(* CODESYS project TC_lib_v0-0-0-1.library
   Company: RWTH
   Title: Tc_Wilo_LIB
   Placeholder: Tc_Wilo_LIB
   Author: Vonnahme
   Version: 0.0.0.1

Project tree, tasks and I/O mapping:
  libraries: Tc2_Standard, * (Beckhoff Automation GmbH); Tc2_System, * (Beckhoff Automation GmbH); Tc2_TcpIp, * (Beckhoff Automation GmbH); Tc2_Utilities, * (Beckhoff Automation GmbH); Tc3_Interfaces, * (Beckhoff Automation GmbH); Tc3_Module, * (Beckhoff Automation GmbH)
  ADS/
    function block FB_ADS_READ [ST]
    function block FB_ADS_WRITE [ST]
  CAN/
    Definitions/
      data type eBusCommand
      data type eBusControlMode
      data type eEffCommand
      data type SDO_Datapoint
      data type StratosControl
      data type WILO_Stratos
      data type WILO_StratosGiga_IPE
    Stratos/
      function block FB_Stratos_CAN [ST]
    StratosGiga_IPE/
      function block FB_StratosGIGA_IPE [ST]
    function block FB_SDO_READ [ST]
    function block FB_SDO_READ_v0 [ST]
    function block FB_SDO_WRITE [ST]
  Datenlogger/
    Definitions/
      data type Log_Datapoint
      data type Log_Struct_HMI
    FB/
      function block FB_FILE [ST]
      function block FB_FOLDER [ST]
      function block FB_LOGGING [ST]
      function block FB_TIME [ST]
    function block FB_Datenlogger [ST]
  Functions/
    function FUN_ByteArrToString [ST]
    function FUN_DatatypSize [ST]
    function FUN_StringToByteArr [ST]
    function SCALE [ST]
  Timetable/
    DUT/
      data type Struct_TimeTable
    function block FB_TimeTable [ST]
  TypeDef/
    data type Datatyp
  Version/
    global variables Global_Version
*)

// CAN/Definitions/eBusCommand
{attribute 'qualified_only'}
{attribute 'strict'}
TYPE eBusCommand : 
(
	RemoteOn:=97,
	RemoteOff:=96
);
END_TYPE

// CAN/Definitions/eBusControlMode
{attribute 'qualified_only'}
//{attribute 'strict'}
TYPE eBusControlMode : 
(
	nc:=0,
	dpc:=5,
	dpv:=6
);
END_TYPE

// CAN/Definitions/eEffCommand
{attribute 'qualified_only'}
//{attribute 'strict'}
TYPE eEffCommand : 
(
	PumpOn:=1,
	PumpOff:=0,
	RemoteOn:=97,
	RemoteOff:=96
);
END_TYPE

// CAN/Definitions/SDO_Datapoint
TYPE SDO_Datapoint :
STRUCT
	sDatapointNo		:STRING;
	sDescription 		:STRING;
	sValue				:STRING;
	eDatatyp			:Datatyp;
	sUnit				:STRING;
	bReadSuccesfull		:BOOL;
END_STRUCT
END_TYPE

// CAN/Definitions/StratosControl
TYPE StratosControl :
STRUCT
		eBusCommand								:eBusCommand;		// PumpOn, PumpOff
		eBusControlMode							:eBusControlMode;	// nc,dpc, dpv
		nBusSetpoint							:LREAL;			//[%,rpm,mWs]
END_STRUCT
END_TYPE

// CAN/Definitions/WILO_Stratos
TYPE WILO_Stratos :
STRUCT
	arrPumpInformation						:ARRAY [1..100] OF SDO_Datapoint;
	iSpeed									:UINT;				//[rpm]	
	nPressure								:LREAL;				//[mWs]
	nFlow									:LREAL;				//[m³/h]		
	nInputPower								:LREAL;				//[W]
	nConsumption							:LREAL;				//[kWh]	
	nMediumTemp								:LREAL;				//[°C]
	nOperatingHours							:LREAL;				//[h]		
	eEff_Command							:eEffCommand;	
	eEff_ControlMode						:eBusControlMode;	
	nEff_Setpoint							:LREAL;				//[%]
	nEff_Setpoint_abs						:LREAL;				//[rpm, mWs]
	eSel_Command							:eEffCommand;
	eSel_ControlMode						:eBusControlMode;	
	nSel_Setpoint							:LREAL;				//[%]
	nSel_Setpoint_abs						:LREAL;				//[rpm, mWs]
	iPumpType								:UINT;				//[PumpType]	
	nMaxValue								:LREAL;				//[mWs], [rpm]
	nMinValue								:LREAL;				//[mWs], [rpm]
	iCurrentWarning							:USINT;				//[Error Code]	
	eBusCommand								:eBusCommand;
	eBusControlMode							:eBusControlMode;
	nBusSetpoint							:LREAL;		
END_STRUCT
END_TYPE

// CAN/Definitions/WILO_StratosGiga_IPE
TYPE WILO_StratosGiga_IPE :
STRUCT
	arrPumpInformation						:ARRAY [1..100] OF SDO_Datapoint;
	iSpeed									:UINT;				//[rpm]	
	nPressure								:LREAL;				//[mWs]
	nFlow									:LREAL;				//[m³/h]		
	nInputPower								:LREAL;				//[W]
	nConsumption							:LREAL;				//[kWh]	
	iPressureSensorSource					:USINT;				// 2 Pump Housing, 3 External, 5 LON
	nOperatingHours							:LREAL;				//[h]		
	eEff_Command							:eEffCommand;	
	eEff_ControlMode						:eBusControlMode;	
	nEff_Setpoint							:LREAL;				//[%]
	nEff_Setpoint_abs						:LREAL;				//[rpm, mWs]
	eSel_Command							:eEffCommand;
	eSel_ControlMode						:eBusControlMode;	
	nSel_Setpoint							:LREAL;				//[%]
	nSel_Setpoint_abs						:LREAL;				//[rpm, mWs]
	iPumpType								:UINT;				//[PumpType]	
	nMaxValue								:LREAL;				//[mWs], [rpm]
	iCurrentWarning							:USINT;				//[Error Code]	
	eBusCommand								:eBusCommand;
	eBusControlMode							:eBusControlMode;
	nBusSetpoint							:LREAL;	
	iBusStatus								:USINT;
	iControlStatus 							:USINT;
	iReadyForOperation 						:USINT;
	iPumpIsOperating 						:USINT;
	iServiceRequired 						:USINT;
	nElectricalCurrent 						:LREAL;				// [A]
	nVoltageLevel 							:LREAL;				// [V]
END_STRUCT
END_TYPE

// Datenlogger/Definitions/Log_Datapoint
TYPE Log_Datapoint :
STRUCT
	sID				:T_MaxString;
	sDescription 	:T_MaxString;
	sUnit			:T_MaxString;
	sValue 			:T_MaxString;
END_STRUCT
END_TYPE

// Datenlogger/Definitions/Log_Struct_HMI
TYPE Log_Struct_HMI :
STRUCT
	bLogging :BOOL;
	sCycleTime :STRING:='T#10s';
	sFolderPath :STRING;
	iErrors	:UINT;
	iNumberOfLoggedDatapoints :INT;
	arrLogDatapoints :ARRAY [0..499] OF Log_Datapoint;
END_STRUCT
END_TYPE

// Timetable/DUT/Struct_TimeTable
TYPE Struct_TimeTable :
STRUCT
	wDayOfWeek	:WORD:=99;		// 0= inactiv, 1=Sunday, 2=Monday, ... 7=Saturday, 8=daily, 9=Weekend, 10=Mo-Fr, 99=last row
	wHour		:WORD;
	wMinute		:WORD;
	nValue		:LREAL;
END_STRUCT
END_TYPE

// TypeDef/Datatyp
{attribute 'qualified_only'}
{attribute 'strict'}
TYPE Datatyp :
(
	_NotDefined:=0,
	_BYTE:=1,
	_WORD:=2,
	_DWORD:=3,
	_SINT:=4,
	_INT:=5,
	_DINT:=6,
	_LINT:=7,
	_USINT:=8,
	_UINT:=9,
	_UDINT:=10,
	_ULINT:=11,
	_REAL:=12,
	_LREAL:=13,
	_BOOL:=14,
	_ENUM:=15
);
END_TYPE

// Version/Global_Version
{attribute 'TcGenerated'}
// This function has been automatically generated from the project information.
VAR_GLOBAL CONSTANT
	{attribute 'const_non_replaced'}
	{attribute 'linkalways'}
	stLibVersion_Tc_Wilo_LIB : ST_LibVersion := (iMajor := 0, iMinor := 0, iBuild := 0, iRevision := 1, sVersion := '0.0.0.1');
END_VAR

// ADS/FB_ADS_READ
FUNCTION_BLOCK FB_ADS_READ
VAR_INPUT
	/// The AMSNetID addresses the FC5101 card. Can be empty if only one local single channel card is present
	ADSNetID: STRING(23);
	/// This Port No. of the Reading DataPoint 
	PortNr: WORD;
	/// hexadecimal '16x000'
	IndexGroup: DWORD;
	/// hexadecimal '16x000'
	IndexOffset: DWORD;
	/// hexadecimal '16x000'
	DataLength: DWORD;
	/// only reset to FALSE after ReadDataAvailable=TRUE
	StartReading: BOOL;
END_VAR
VAR_OUTPUT
	ReadData: ARRAY[0..255] OF BYTE;
	ReadDataAvailable: BOOL;
	Error: DWORD;
END_VAR
VAR
	state: BYTE := 0;
	ADSREAD: ADSREAD;
END_VAR

CASE state OF
0:
	IF StartReading THEN
		ReadDataAvailable := FALSE;
		Error := 0;
		ADSRead(
			NETID:= ADSNetID,
			PORT:= PortNr,
			IDXGRP:= IndexGroup,
			IDXOFFS:= IndexOffset,
			LEN:= DataLength,
			DESTADDR:= ADR(ReadData),
			READ:= TRUE,
			TMOUT := T#1s
		);
		IF ADSRead.err THEN
			state := 2;
			(*ReadDataAvailable := TRUE;*)
			Error := ADSRead.ErrId;
		ELSE
			state := 1;
		END_IF
	ELSE
		ADSRead(
			NETID:= ADSNetID,
			PORT:= PortNr,
			IDXGRP:= IndexGroup,
			IDXOFFS:= IndexOffset,
			LEN:= DataLength,
			DESTADDR:= ADR(ReadData),
			READ:= FALSE,
			TMOUT := T#1s
		);
	END_IF

1:
	ADSRead(READ:= FALSE);
	IF ADSRead.err THEN
		state := 2;
		(*ReadDataAvailable := TRUE;*)
		Error := ADSRead.ErrId;
	ELSE
		IF NOT ADSRead.busy THEN
			state := 2;
			(*ReadDataAvailable := TRUE;*)
		END_IF
	END_IF

2: 
	ADSRead(READ:= FALSE);
	ReadDataAvailable := TRUE;
	state := 0;
END_CASE

END_FUNCTION_BLOCK

// ADS/FB_ADS_WRITE
FUNCTION_BLOCK FB_ADS_WRITE
VAR_INPUT
	/// The AMSNetID addresses the FC5101 card. Can be empty if only one local single channel card is present
	ADSNetID: STRING(23);
	/// This Port No. of the Reading DataPoint 
	PortNr: WORD;
	/// hexadecimal '16x000'
	IndexGroup: DWORD;
	/// hexadecimal '16x000'
	IndexOffset: DWORD;
	/// hexadecimal '16x000'
	DataLength: DWORD;
	/// only reset to FALSE after WriteDataFinished=TRUE
	StartWriting: BOOL;
	///This array contains the data to be written to the CANopen Object Dictionary
	WriteData: ARRAY[0..255] OF BYTE;
END_VAR
VAR_OUTPUT
	WriteDataFinished: BOOL;
	Error: DWORD;
END_VAR
VAR
	state: BYTE := 0;
	ADSWRITE: ADSWRITE;
END_VAR

CASE state OF
0:
	IF StartWriting THEN
		WriteDataFinished := FALSE;
		Error := 0;
		ADSWrite(
			NETID:= ADSNetID,
			PORT:= PortNr,
			IDXGRP:= IndexGroup,
			IDXOFFS:= IndexOffset,
			LEN:= DataLength,
			SRCADDR:= ADR(WriteData),
			WRITE:= TRUE,
			TMOUT := T#1s
		);
		IF ADSWrite.err THEN
			state := 2;
			(*WriteDataFinished := TRUE;*)
			Error := ADSWrite.ErrId;
		ELSE
			state := 1;
		END_IF
	ELSE
		ADSWrite(
			NETID:= '',
			PORT:= PortNr,
			IDXGRP:= IndexGroup,
			IDXOFFS:= IndexOffset,
			LEN:= DataLength,
			SRCADDR:= ADR(WriteData),
			WRITE:= FALSE,
			TMOUT := T#1s
		);
	END_IF

1:
	ADSWrite(WRITE:= FALSE);
	IF ADSWrite.err THEN
		state := 2;
		(*WriteDataFinished := TRUE;*)
		Error := ADSWrite.ErrId;
	ELSE
		IF NOT ADSWrite.busy THEN
			state := 2;
			(*WriteDataFinished := TRUE;*)
		END_IF
	END_IF

2:
	ADSWrite(WRITE:= FALSE);
	state := 0;
	WriteDataFinished := TRUE;
END_CASE

END_FUNCTION_BLOCK

// CAN/Stratos/FB_Stratos_CAN
FUNCTION_BLOCK FB_Stratos_CAN
VAR_INPUT
	// CAN configuration
		sCAN_NetID								:STRING (23);	// NetID of CAN Master
		iCAN_NodeID								:UINT;		// NodeId (automatic calculation of Port No.
	// control configuration
		bReadOnly								:BOOL;		// deactivate pump control
		bUseAbsoluteSetpoint					:BOOL;		// use rpm or mWs instead of %
		bExternalCommandOverride				:BOOL:=TRUE;	// Use  for pump control Struct instead of PumpInformationStruct to control the pump
		stPumpControl							:StratosControl; // Struct for control pump by external PLC Code
END_VAR
VAR_OUTPUT
	// Error
		iReadError								:UINT;	// number of Errors (read)
		iWriteError								:UINT;	// number of Errors (write)
	
	// Structure	
		stPumpInformation						:WILO_Stratos; // Information (Control) of pump
			
	// Logging
		arrDatenpunkt_IDs_Pump					:ARRAY [0..99] OF T_MaxString;			(*Beschreibung der Datenpunkte*)
		arrDatenpunkt_Values_Pump				:ARRAY [0..99] OF T_MaxString;			(*Messwerte der Datenpunkte*)
		iDatapoints_Pump						:INT			:=0;
END_VAR
VAR	
	// Datapoints
(*		iSpeed									:UINT;			//[rpm]	
		nPressure								:LREAL;			//[mWs]
		nFlow									:LREAL;			//[m³/h]		
		nInputPower								:LREAL;			//[W]
		nConsumption							:LREAL;			//[kWh]	
		nMediumTemp								:LREAL;			//[°C]
		nOperatingHours							:LREAL;			//[h]		
		eEff_Command							:eEffCommand;	
		eEff_ControlMode						:eBusControlMode;	
		nEff_Setpoint							:LREAL;			//[%]
		nEff_Setpoint_abs						:LREAL;			//[rpm, mWs]
		eSel_Command							:eEffCommand;
		eSel_ControlMode						:eBusControlMode;
		nSel_Setpoint							:LREAL;			//[%]
		nSel_Setpoint_abs						:LREAL;			//[rpm, mWs]
		iPumpType								:UINT;			//[PumpType]	
		nMaxValue								:LREAL;			//[mWs], [rpm]
		iCurrentWarning							:USINT;			//[Error Code]		
*)
	// Read
		imaxValue								:UINT;	
		iminValue								:UINT;	
		iInputPower								:UDINT;	
		iPressure								:UINT;		
		iMediumTemp								:UINT;			
		iFlow									:UINT;	
		ieff_Setpoint							:INT;					
		iEff_ControlMode					 	:USINT;
		ieff_Command							:USINT;	
		iSel_Setpoint							:INT;					
		iSel_ControlMode					 	:USINT;
		iSel_Command							:USINT;
		iConsumption							:UDINT;	
		iOperatingHours							:UDINT;			
		
	// Write
		iBusCommand								:USINT;			//16#61=PumpOn; 16#60=PumpOff
		iBusControlMode					 		:USINT;			//0=nc; 5=dpc; 6=dpv
		iBusSetpoint					 		:INT;			
	
	// CAN
		State_CAN								:INT		:=0;	
	
	// CAN-ini
		CAN_NodePort							:WORD;
		
	// CAN-Datenpunkteigenschaften
		CAN_Index								:DWORD;
		CAN_Subindex							:DWORD;
		CAN_Length								:DWORD;
		CAN_RW_Mode								:INT		:=0;
		CAN_Start								:BOOL		:=FALSE;
		iDpAddres								:POINTER TO ARRAY [0..7] OF BYTE;
		bReadSuccesfull							:BOOL;
		
	// CAN-SDO_Write Baustein
		CAN_SDO_WRITE							:FB_SDO_WRITE;
		CAN_WriteData							:ARRAY[0..255] OF BYTE;
		CAN_WriteError							:DWORD;
		
	// CAN-SDO_Read Baustein
		CAN_SDO_READ							:FB_SDO_READ;
		CAN_ReadData							:ARRAY[0..255] OF BYTE;
		CAN_ReadError							:DWORD;
		CAN_ScaleNum							:REAL			:=1;
		CAN_ScaleDenum							:REAL			:=1;
		CAN_ScaleOffset							:REAL			:=0;	
		CAN_Description							:STRING;
		CAN_Datatype							:Datatyp;
		CAN_Unit								:STRING;
		CAN_Unit_abs							:STRING;
END_VAR

// calculate NodePort by NodeID
CAN_NodePort:=16#1000+iCAN_NodeID;	

IF bExternalCommandOverride THEN
	stPumpInformation.eBusCommand:= stPumpControl.eBusCommand;
	stPumpInformation.eBusControlMode:= stPumpControl.eBusControlMode;
	stPumpInformation.nBusSetpoint:= stPumpControl.nBusSetpoint;
END_IF

// SDO-Pumpendatenpunkte	
	CASE State_CAN OF
	0:  // Initialisierung
		State_CAN := 1;
		
	1:	// Datenpunkt Pump Type
		CAN_Index:=16#2182;
		CAN_Subindex:=16#1;
		CAN_Length:=16#2;
		CAN_RW_Mode:=1;
		CAN_ScaleNum:=1;
		CAN_ScaleDenum:=1;
		CAN_ScaleOffset:=0;
		CAN_Description:='PumpType';
		CAN_Unit:='-';
		CAN_Datatype:=9;
		iDpAddres:=ADR(stPumpInformation.iPumpType);
		
		IF bReadSuccesfull THEN
			stPumpinformation.arrPumpInformation[State_CAN].sValue:=UINT_TO_STRING(stPumpInformation.iPumpType);
			bReadSuccesfull:=FALSE;
			State_CAN := State_CAN+1;
		END_IF
		
	2:	// Datenpunkt maxFörderhöhe [mWs] bzw. maxDrehzahl [rpm]
		CASE ieff_ControlMode OF
			0:		CAN_Index:=16#21A1;
					CAN_ScaleNum:=1;
					CAN_ScaleDenum:=1;
					CAN_ScaleOffset:=0;
					CAN_Unit:='rpm';
					CAN_Unit_abs:='rpm';
					
			5:		CAN_Index:=16#21AD;
					CAN_ScaleNum:=102;
					CAN_ScaleDenum:=10000;
					CAN_ScaleOffset:=0;
					CAN_Unit:='mWs';
					CAN_Unit_abs:='mWs';
			
			6:		CAN_Index:=16#21A5;
					CAN_ScaleNum:=102;
					CAN_ScaleDenum:=10000;
					CAN_ScaleOffset:=0;
					CAN_Unit:='mWs';
					CAN_Unit_abs:='mWs';
			
			ELSE	CAN_Index:=16#21AD;
					CAN_ScaleNum:=102;
					CAN_ScaleDenum:=10000;
					CAN_ScaleOffset:=0;
					CAN_Unit:='mWs';	
					CAN_Unit_abs:='mWs';	
		END_CASE
		
		CAN_Subindex:=16#0;
		CAN_Length:=16#2;	
		CAN_RW_Mode:=1;
		CAN_Description:='maxValue';
		CAN_Datatype:=13;
		iDpAddres:=ADR(imaxValue);
		
		IF bReadSuccesfull THEN
			stPumpInformation.nmaxValue:=SCALE(imaxValue,CAN_ScaleNum,CAN_ScaleDenum,CAN_ScaleOffset);			
			stPumpinformation.arrPumpInformation[State_CAN].sValue:=LREAL_TO_STRING(stPumpInformation.nMaxValue);
			bReadSuccesfull:=FALSE;			
			State_CAN := State_CAN+1;
		END_IF

	3:	// Datenpunkt Speed [rpm]
		CAN_Index:=16#2083;
		CAN_Subindex:=16#1;
		CAN_Length:=16#2;
		CAN_RW_Mode:=1;
		CAN_ScaleNum:=1;
		CAN_ScaleDenum:=1;
		CAN_ScaleOffset:=0;
		CAN_Description:='Speed';
		CAN_Unit:='rpm';
		CAN_Datatype:=9;
		iDpAddres:=ADR(stPumpInformation.ispeed);
		
		IF bReadSuccesfull THEN
			stPumpinformation.arrPumpInformation[State_CAN].sValue:=UINT_TO_STRING(stPumpInformation.ispeed);
			bReadSuccesfull:=FALSE;	
			State_CAN := State_CAN+1;
		END_IF
		
	4:	// Datenpunkt Flow [m^3/h]
		CAN_Index:=16#2087;
		CAN_Subindex:=16#0;
		CAN_Length:=16#2;
		CAN_RW_Mode:=1;
		CAN_ScaleNum:=1;
		CAN_ScaleDenum:=10;
		CAN_ScaleOffset:=0;
		CAN_Description:='EstimatedFlow';
		CAN_Unit:='m³/h';
		CAN_Datatype:=13;
		iDpAddres:=ADR(iflow);
		
		IF bReadSuccesfull THEN
			stPumpInformation.nflow:=SCALE(iflow,CAN_ScaleNum,CAN_ScaleDenum,CAN_ScaleOffset);
			stPumpinformation.arrPumpInformation[State_CAN].sValue:=LREAL_TO_STRING(stPumpInformation.nflow);
			bReadSuccesfull:=FALSE;	
			State_CAN := State_CAN+1;
		END_IF
			
	5:	// Datenpunkt Consumption [kWh]
		CAN_Index:=16#2113;
		CAN_Subindex:=16#0;
		CAN_Length:=16#4;
		CAN_RW_Mode:=1;
		CAN_ScaleNum:=1;
		CAN_ScaleDenum:=10;
		CAN_ScaleOffset:=0;
		CAN_Description:='Consumption';
		CAN_Unit:='kWh';
		CAN_Datatype:=13;
		iDpAddres:=ADR(iConsumption);
		
		IF bReadSuccesfull THEN
			stPumpInformation.nConsumption:=SCALE(iConsumption,CAN_ScaleNum,CAN_ScaleDenum,CAN_ScaleOffset);
			stPumpinformation.arrPumpInformation[State_CAN].sValue:=LREAL_TO_STRING(stPumpInformation.nConsumption);
			bReadSuccesfull:=FALSE;	
			State_CAN := State_CAN+1;		
		END_IF
	
	6:	// Datenpunkt Operating Hours [h]
		CAN_Index:=16#2101;
		CAN_Subindex:=16#0;
		CAN_Length:=16#4;
		CAN_RW_Mode:=1;
		CAN_ScaleNum:=1;
		CAN_ScaleDenum:=60;
		CAN_ScaleOffset:=0;
		CAN_Description:='OperationTimeResettable';
		CAN_Unit:='kWh';
		CAN_Datatype:=13;
		iDpAddres:=ADR(iOperatingHours);
		
		IF bReadSuccesfull THEN
			stPumpInformation.nOperatingHours:=SCALE(iOperatingHours,CAN_ScaleNum,CAN_ScaleDenum,CAN_ScaleOffset);			
			stPumpinformation.arrPumpInformation[State_CAN].sValue:=LREAL_TO_STRING(stPumpInformation.nOperatingHours);
			bReadSuccesfull:=FALSE;	
			State_CAN := State_CAN+1;
		END_IF
		
	7:	// Datenpunkt Current Warning
		CAN_Index:=16#20C1;
		CAN_Subindex:=16#0;
		CAN_Length:=16#1;
		CAN_RW_Mode:=1;
		CAN_ScaleNum:=1;
		CAN_ScaleDenum:=1;
		CAN_ScaleOffset:=0;
		CAN_Description:='CurrentWarning_Error';
		CAN_Unit:='-';
		CAN_Datatype:=8;
		iDpAddres:=ADR(stPumpInformation.iCurrentWarning);
		
		IF bReadSuccesfull THEN
			stPumpinformation.arrPumpInformation[State_CAN].sValue:=USINT_TO_STRING(stPumpInformation.iCurrentWarning);
			bReadSuccesfull:=FALSE;	
			State_CAN := State_CAN+1;
		END_IF
		
	8: 	// Datenpunkt Input Power
		CAN_Index:=16#2090;
		CAN_Subindex:=16#0;
		CAN_Length:=16#4;
		CAN_RW_Mode:=1;
		CAN_ScaleNum:=1;
		CAN_ScaleDenum:=1000;
		CAN_ScaleOffset:=0;
		CAN_Description:='InputPower';
		CAN_Unit:='W';
		CAN_Datatype:=13;
		iDpAddres:=ADR(iInputPower);
		
		IF bReadSuccesfull THEN
			stPumpInformation.nInputPower:=SCALE(iInputPower,CAN_ScaleNum,CAN_ScaleDenum,CAN_ScaleOffset);
			stPumpinformation.arrPumpInformation[State_CAN].sValue:=LREAL_TO_STRING(stPumpInformation.nInputPower);
			bReadSuccesfull:=FALSE;	
			State_CAN := State_CAN+1;
		END_IF
		
	9: 	// Datenpunkt Estimated Pressure
		CAN_Index:=16#208B;
		CAN_Subindex:=16#0;
		CAN_Length:=16#2;
		CAN_RW_Mode:=1;
		CAN_ScaleNum:=102;
		CAN_ScaleDenum:=10000;
		CAN_ScaleOffset:=0;
		CAN_Description:='Estimated Pressure';
		CAN_Unit:='mWs';
		CAN_Datatype:=13;
		iDpAddres:=ADR(iPressure);
		
		IF bReadSuccesfull THEN
			stPumpInformation.nPressure:=SCALE(iPressure,CAN_ScaleNum,CAN_ScaleDenum,CAN_ScaleOffset);
			stPumpinformation.arrPumpInformation[State_CAN].sValue:=LREAL_TO_STRING(stPumpInformation.nPressure);
			bReadSuccesfull:=FALSE;	
			State_CAN := State_CAN+1;
		END_IF
		
	10: // Datenpunkt Medium Temperature
		CAN_Index:=16#20A0;
		CAN_Subindex:=16#0;
		CAN_Length:=16#2;
		CAN_RW_Mode:=1;
		CAN_ScaleNum:=1;
		CAN_ScaleDenum:=10;
		CAN_ScaleOffset:=-273.15;
		CAN_Description:='MediumTemperature';
		CAN_Unit:='°C';
		CAN_Datatype:=13;
		iDpAddres:=ADR(iMediumTemp);
		
		IF bReadSuccesfull THEN
			stPumpInformation.nMediumTemp:=SCALE(UINT_TO_LREAL(iMediumTemp),CAN_ScaleNum,CAN_ScaleDenum,CAN_ScaleOffset);
			stPumpinformation.arrPumpInformation[State_CAN].sValue:=LREAL_TO_STRING(stPumpInformation.nMediumTemp);
			bReadSuccesfull:=FALSE;	
			State_CAN := State_CAN+1;
		END_IF
		
	11: // Datenpunkt effective Capacity
		CAN_Index:=16#2040;
		CAN_Subindex:=16#0;
		CAN_Length:=16#2;
		CAN_RW_Mode:=1;
		CAN_ScaleNum:=1;
		CAN_ScaleDenum:=100;
		CAN_ScaleOffset:=0;
		CAN_Description:='Effective Capacity';
		CAN_Unit:='%';
		CAN_Datatype:=13;
		iDpAddres:=ADR(ieff_Setpoint);
		
		IF bReadSuccesfull THEN
			stPumpInformation.neff_Setpoint:=SCALE(ieff_Setpoint,CAN_ScaleNum,CAN_ScaleDenum,CAN_ScaleOffset);
			stPumpInformation.neff_Setpoint_abs:=stPumpInformation.neff_Setpoint/100*stPumpInformation.nMaxValue;
			IF bUseAbsoluteSetpoint THEN
				stPumpinformation.arrPumpInformation[State_CAN].sValue:=LREAL_TO_STRING(stPumpInformation.neff_Setpoint_abs);
				stPumpinformation.arrPumpInformation[State_CAN].sUnit:=CAN_Unit_abs;	
			ELSE
				stPumpinformation.arrPumpInformation[State_CAN].sValue:=LREAL_TO_STRING(stPumpInformation.neff_Setpoint);
			END_IF
			bReadSuccesfull:=FALSE;	
			State_CAN := State_CAN+1;
		END_IF
				
	12: // Datenpunkt effective Control Mode
		CAN_Index:=16#2041;
		CAN_Subindex:=16#0;
		CAN_Length:=16#1;
		CAN_RW_Mode:=1;
		CAN_ScaleNum:=1;
		CAN_ScaleDenum:=1;
		CAN_ScaleOffset:=0;
		CAN_Description:='EffectiveControlMode';
		CAN_Unit:='-';
		CAN_Datatype:=15;
		iDpAddres:=ADR(ieff_ControlMode);
		
		IF bReadSuccesfull THEN
			stPumpInformation.eeff_ControlMode:=USINT_TO_INT(ieff_ControlMode);
			stPumpinformation.arrPumpInformation[State_CAN].sValue:=USINT_TO_STRING(ieff_ControlMode);
			bReadSuccesfull:=FALSE;	
			State_CAN := State_CAN+1;
		END_IF

	13: // Datenpunkt effective Command
		CAN_Index:=16#2042;
		CAN_Subindex:=16#0;
		CAN_Length:=16#1;
		CAN_RW_Mode:=1;
		CAN_ScaleNum:=1;
		CAN_ScaleDenum:=1;
		CAN_ScaleOffset:=0;
		CAN_Description:='EffectiveCommand';
		CAN_Unit:='-';
		CAN_Datatype:=15;
		iDpAddres:=ADR(ieff_Command);
		
		IF bReadSuccesfull THEN
			stPumpInformation.eeff_Command:=USINT_TO_INT(ieff_Command);
			stPumpinformation.arrPumpInformation[State_CAN].sValue:=USINT_TO_STRING(ieff_Command);
			bReadSuccesfull:=FALSE;	
			State_CAN := State_CAN+1;
		END_IF

	14: // Datenpunkt Selected BusSetpoint
		CAN_Index:=16#2048;
		CAN_Subindex:=16#0;
		CAN_Length:=16#2;
		CAN_RW_Mode:=1;
		CAN_ScaleNum:=1;
		CAN_ScaleDenum:=100;
		CAN_ScaleOffset:=0;
		CAN_Description:='SelectedSetpoint';
		CAN_Unit:='%';
		CAN_Datatype:=13;
		iDpAddres:=ADR(iSel_Setpoint);
		
		IF bReadSuccesfull THEN
			stPumpInformation.nSel_Setpoint:=SCALE(iSel_Setpoint,CAN_ScaleNum,CAN_ScaleDenum,CAN_ScaleOffset);
			stPumpInformation.nSel_Setpoint_abs:=stPumpInformation.nSel_Setpoint/100*stPumpInformation.nMaxValue;
			IF bUseAbsoluteSetpoint THEN
				stPumpinformation.arrPumpInformation[State_CAN].sValue:=LREAL_TO_STRING(stPumpInformation.nSel_Setpoint_abs);
				stPumpinformation.arrPumpInformation[State_CAN].sUnit:=CAN_Unit_abs;	
			ELSE
				stPumpinformation.arrPumpInformation[State_CAN].sValue:=LREAL_TO_STRING(stPumpInformation.nSel_Setpoint);
			END_IF		
			bReadSuccesfull:=FALSE;	
			State_CAN := State_CAN+1;
		END_IF
		
	15:	// Datenpunkt Selected Control Mode
		CAN_Index:=16#2049;
		CAN_Subindex:=16#0;
		CAN_Length:=16#1;
		CAN_RW_Mode:=1;
		CAN_ScaleNum:=1;
		CAN_ScaleDenum:=1;
		CAN_ScaleOffset:=0;
		CAN_Description:='SelectedControlMode';
		CAN_Unit:='-';
		CAN_Datatype:=15;
		iDpAddres:=ADR(iSel_ControlMode);
		
		IF bReadSuccesfull THEN
			stPumpInformation.eSel_ControlMode:=USINT_TO_INT(iSel_ControlMode);
			stPumpinformation.arrPumpInformation[State_CAN].sValue:=USINT_TO_STRING(iSel_ControlMode);
			bReadSuccesfull:=FALSE;	
			State_CAN := State_CAN+1;
		END_IF
		
	16:	// Datenpunkt Selected BusCommand
		CAN_Index:=16#204A;
		CAN_Subindex:=16#0;
		CAN_Length:=16#1;
		CAN_RW_Mode:=1;
		CAN_ScaleNum:=1;
		CAN_ScaleDenum:=1;
		CAN_ScaleOffset:=0;
		CAN_Description:='Selected Command';
		CAN_Unit:='-';
		CAN_Datatype:=15;
		iDpAddres:=ADR(iSel_Command);
		
		IF bReadSuccesfull THEN
			stPumpInformation.eSel_Command:=USINT_TO_INT(iSel_Command);
			stPumpinformation.arrPumpInformation[State_CAN].sValue:=USINT_TO_STRING(iSel_Command);
			bReadSuccesfull:=FALSE;	
			State_CAN := State_CAN+1;
		END_IF

	17:	// Datenpunkt BusCommand
		iBusCommand:=INT_TO_USINT(stPumpInformation.eBusCommand);
		
		CAN_Index:=16#200A;
		CAN_Subindex:=16#0;
		CAN_Length:=16#1;
		CAN_RW_Mode:=2;
		
		MEMCPY(ADR(CAN_WriteData),ADR(iBusCommand),CAN_Length);
	
	18: // Datenpunkt BusControlMode
		iBusControlMode:=INT_TO_USINT(stPumpInformation.eBusControlMode);

		CAN_Index:=16#2009;
		CAN_Subindex:=16#0;
		CAN_Length:=16#1;
		CAN_RW_Mode:=2;
		
		MEMCPY(ADR(CAN_WriteData),ADR(iBusControlMode),CAN_Length);	
		
	19: // Datenpunkt BusSetpoint
		CAN_Index:=16#2008;
		CAN_Subindex:=16#0;
		CAN_Length:=16#2;
		CAN_RW_Mode:=2;		

		IF bUseAbsoluteSetpoint AND imaxValue<>0 THEN
			iBusSetpoint:=LREAL_TO_INT (SCALE(stPumpInformation.nBusSetpoint/stPumpInformation.nmaxValue*100,100,1,0));
		ELSE
			iBusSetpoint:=LREAL_TO_INT (SCALE(stPumpInformation.nBusSetpoint,100,1,0));
		END_IF
				
		MEMCPY(ADR(CAN_WriteData),ADR(iBusSetpoint),CAN_Length);
	
	20:	// Datenpunkt minFörderhöhe [mWs] bzw. minDrehzahl [rpm]
		CASE ieff_ControlMode OF
			0:		CAN_Index:=16#21A0;
					CAN_ScaleNum:=1;
					CAN_ScaleDenum:=1;
					CAN_ScaleOffset:=0;
					CAN_Unit:='rpm';
					CAN_Unit_abs:='rpm';
					
			5:		CAN_Index:=16#21AC;
					CAN_ScaleNum:=102;
					CAN_ScaleDenum:=10000;
					CAN_ScaleOffset:=0;
					CAN_Unit:='mWs';
					CAN_Unit_abs:='mWs';
			
			6:		CAN_Index:=16#21A4;
					CAN_ScaleNum:=102;
					CAN_ScaleDenum:=10000;
					CAN_ScaleOffset:=0;
					CAN_Unit:='mWs';
					CAN_Unit_abs:='mWs';
			
			ELSE	CAN_Index:=16#21AD;
					CAN_ScaleNum:=102;
					CAN_ScaleDenum:=10000;
					CAN_ScaleOffset:=0;
					CAN_Unit:='mWs';	
					CAN_Unit_abs:='mWs';	
		END_CASE
		
		CAN_Subindex:=16#0;
		CAN_Length:=16#2;	
		CAN_RW_Mode:=1;
		CAN_Description:='minValue';
		CAN_Datatype:=13;
		iDpAddres:=ADR(iminValue);
		
		IF bReadSuccesfull THEN
			stPumpInformation.nminValue:=SCALE(iminValue,CAN_ScaleNum,CAN_ScaleDenum,CAN_ScaleOffset);			
			stPumpinformation.arrPumpInformation[State_CAN].sValue:=LREAL_TO_STRING(stPumpInformation.nMinValue);
			bReadSuccesfull:=FALSE;			
			State_CAN := State_CAN+1;
		END_IF
	
	21: // Step to First DP
		State_CAN := 1;
	END_CASE
	
// SDO_Datenpunkte lesen/schreiben
	CASE CAN_RW_Mode OF
	0:  // Bausteine nicht ausführen		
	1:	// SDO_Read
		CAN_SDO_READ(
			StartReading := CAN_Start,
			CO_Index := 	CAN_Index,
			CO_SubIndex := 	CAN_Subindex,
			DataLength := 	CAN_Length,
			PortNr := 		CAN_NodePort,
			ADSNetID :=		sCAN_NetID,
(*			ScaleNum :=		CAN_ScaleNum,
			ScaleDenum := 	CAN_ScaleDenum,
			ScaleOffset := 	CAN_ScaleOffset*)
			);
			
		IF CAN_Start THEN
			IF CAN_SDO_READ.ReadDataAvailable THEN
				CAN_ReadError := CAN_SDO_READ.Error;
				IF CAN_SDO_READ.Error<>0  THEN
					iReadError:=iReadError+1;
					stPumpinformation.arrPumpInformation[State_CAN].bReadSuccesfull:=FALSE;
					stPumpinformation.arrPumpInformation[State_CAN].sDatapointNo:=CONCAT (DWORD_TO_HEXSTR(CAN_Index,2,FALSE),CONCAT('_',DWORD_TO_HEXSTR(CAN_Subindex,2,FALSE)));
					stPumpinformation.arrPumpInformation[State_CAN].sDescription:=CAN_Description;
					stPumpinformation.arrPumpInformation[State_CAN].sUnit:=CAN_Unit;	
					stPumpinformation.arrPumpInformation[State_CAN].eDatatyp:=CAN_Datatype;
					State_CAN := State_CAN+1;
				ELSE
					CAN_ReadData := CAN_SDO_READ.ReadData;
					MEMCPY(iDpAddres,ADR(CAN_ReadData),CAN_Length);
					stPumpinformation.arrPumpInformation[State_CAN].bReadSuccesfull:=TRUE;
					stPumpinformation.arrPumpInformation[State_CAN].sDatapointNo:=CONCAT (DWORD_TO_HEXSTR(CAN_Index,2,FALSE),CONCAT('_',DWORD_TO_HEXSTR(CAN_Subindex,2,FALSE)));
					stPumpinformation.arrPumpInformation[State_CAN].sDescription:=CAN_Description;
					stPumpinformation.arrPumpInformation[State_CAN].sUnit:=CAN_Unit;		
					stPumpinformation.arrPumpInformation[State_CAN].eDatatyp:=CAN_Datatype;				
					bReadSuccesfull:=TRUE;	
				END_IF		
				CAN_Start := FALSE;
				CAN_RW_Mode:=0;
			END_IF
		ELSE
			CAN_Start:=TRUE;
		END_IF

			
	2: 	// SDO_Write
		IF bReadOnly THEN
			State_CAN := 1;
			CAN_Start:=FALSE;
		ELSE
			CAN_SDO_WRITE(
				StartWriting := CAN_Start,
				CO_Index := 	CAN_Index,
				CO_SubIndex := 	CAN_Subindex,
				DataLength := 	CAN_Length,
				PortNr := 		CAN_NodePort,
				ADSNetID:=		sCAN_NetID,
				WriteData:= 	CAN_WriteData
				);			
			IF CAN_Start THEN
				IF CAN_SDO_WRITE.WriteDataFinished THEN
					CAN_WriteError := CAN_SDO_WRITE.Error;
					IF CAN_SDO_Write.Error<>0  THEN
						iWriteError:=iWriteError+1;
					END_IF
					CAN_Start := FALSE;
					State_CAN := State_CAN+1;
				END_IF
			ELSE
				CAN_Start:=TRUE;
			END_IF
		END_IF			
	END_CASE

// Structure
	(*stPumpInformation.iSpeed:= iSpeed;
	stPumpInformation.nPressure:= nPressure;
	stPumpInformation.nFlow:= nFlow;
	stPumpInformation.nInputPower:= nInputPower;
	stPumpInformation.nConsumption:= nConsumption;
	stPumpInformation.nMediumTemp:= nMediumTemp;
	stPumpInformation.nOperatingHours:= nOperatingHours;
	stPumpInformation.eEff_Command:= eEff_Command;
	stPumpInformation.eEff_ControlMode:= eEff_ControlMode;
	stPumpInformation.nEff_Setpoint:= nEff_Setpoint;
	stPumpInformation.nEff_Setpoint_abs:= nEff_Setpoint_abs;
	stPumpInformation.eSel_Command:=eSel_Command;							
	stPumpInformation.eSel_ControlMode:=eSel_ControlMode;							
	stPumpInformation.nSel_Setpoint:=nSel_Setpoint;
	stPumpInformation.nSel_Setpoint_abs:=nSel_Setpoint_abs;					
	stPumpInformation.iPumpType:= iPumpType;
	stPumpInformation.nMaxValue:= nMaxValue;
	stPumpInformation.iCurrentWarning:= iCurrentWarning;*)


// Write Datapoints to LogArray
	iDatapoints_Pump:=0;
	arrDatenpunkt_IDs_Pump[iDatapoints_Pump]:='iSpeed	[rpm]';
	arrDatenpunkt_Values_Pump[iDatapoints_Pump]:=UINT_TO_STRING(stPumpInformation.iSpeed);
	iDatapoints_Pump:=iDatapoints_Pump+1;
		
	arrDatenpunkt_IDs_Pump[iDatapoints_Pump]:='nPressure	[mWs]';
	arrDatenpunkt_Values_Pump[iDatapoints_Pump]:=LREAL_TO_FMTSTR(stPumpInformation.nPressure,2,TRUE);
	iDatapoints_Pump:=iDatapoints_Pump+1;

	arrDatenpunkt_IDs_Pump[iDatapoints_Pump]:='nFlow	[m³/h]';
	arrDatenpunkt_Values_Pump[iDatapoints_Pump]:=LREAL_TO_FMTSTR(stPumpInformation.nFlow,1,TRUE);
	iDatapoints_Pump:=iDatapoints_Pump+1;		
	
	arrDatenpunkt_IDs_Pump[iDatapoints_Pump]:='nInputPower	[W]';
	arrDatenpunkt_Values_Pump[iDatapoints_Pump]:=LREAL_TO_FMTSTR(stPumpInformation.nInputPower,1,TRUE);
	iDatapoints_Pump:=iDatapoints_Pump+1;
	
	arrDatenpunkt_IDs_Pump[iDatapoints_Pump]:='nConsumption	[kWh]';
	arrDatenpunkt_Values_Pump[iDatapoints_Pump]:=LREAL_TO_FMTSTR(stPumpInformation.nConsumption,0,TRUE);
	iDatapoints_Pump:=iDatapoints_Pump+1;
	
	arrDatenpunkt_IDs_Pump[iDatapoints_Pump]:='nMediumTemp	[°C]';
	arrDatenpunkt_Values_Pump[iDatapoints_Pump]:=LREAL_TO_FMTSTR(stPumpInformation.nMediumTemp,2,TRUE);
	iDatapoints_Pump:=iDatapoints_Pump+1;
	
	arrDatenpunkt_IDs_Pump[iDatapoints_Pump]:='nOperatingHours	[h]';
	arrDatenpunkt_Values_Pump[iDatapoints_Pump]:=LREAL_TO_FMTSTR(stPumpInformation.nOperatingHours,0,TRUE);
	iDatapoints_Pump:=iDatapoints_Pump+1;
	
	arrDatenpunkt_IDs_Pump[iDatapoints_Pump]:='eEff_Command	[]';
	arrDatenpunkt_Values_Pump[iDatapoints_Pump]:=INT_TO_STRING(stPumpInformation.eEff_Command);
	iDatapoints_Pump:=iDatapoints_Pump+1;
	
	arrDatenpunkt_IDs_Pump[iDatapoints_Pump]:='eEff_ControlMode	[]';
	arrDatenpunkt_Values_Pump[iDatapoints_Pump]:=INT_TO_STRING(stPumpInformation.eEff_ControlMode);
	iDatapoints_Pump:=iDatapoints_Pump+1;
	
	arrDatenpunkt_IDs_Pump[iDatapoints_Pump]:='nEff_Setpoint	[%]';
	arrDatenpunkt_Values_Pump[iDatapoints_Pump]:=LREAL_TO_FMTSTR(stPumpInformation.nEff_Setpoint,2,TRUE);
	iDatapoints_Pump:=iDatapoints_Pump+1;
	
	arrDatenpunkt_IDs_Pump[iDatapoints_Pump]:='nEff_Setpoint_abs	[rpm, mWs]';
	arrDatenpunkt_Values_Pump[iDatapoints_Pump]:=LREAL_TO_FMTSTR(stPumpInformation.nEff_Setpoint_abs,2,TRUE);
	iDatapoints_Pump:=iDatapoints_Pump+1;

	arrDatenpunkt_IDs_Pump[iDatapoints_Pump]:='eSel_Command	[]';
	arrDatenpunkt_Values_Pump[iDatapoints_Pump]:=INT_TO_STRING(stPumpInformation.eSel_Command);
	iDatapoints_Pump:=iDatapoints_Pump+1;
	
	arrDatenpunkt_IDs_Pump[iDatapoints_Pump]:='eSel_ControlMode	[]';
	arrDatenpunkt_Values_Pump[iDatapoints_Pump]:=INT_TO_STRING(stPumpInformation.eSel_ControlMode);
	iDatapoints_Pump:=iDatapoints_Pump+1;
	
	arrDatenpunkt_IDs_Pump[iDatapoints_Pump]:='nSel_Setpoint	[%]';
	arrDatenpunkt_Values_Pump[iDatapoints_Pump]:=LREAL_TO_FMTSTR(stPumpInformation.nSel_Setpoint,2,TRUE);
	iDatapoints_Pump:=iDatapoints_Pump+1;
	
	arrDatenpunkt_IDs_Pump[iDatapoints_Pump]:='nSel_Setpoint_abs	[rpm, mWs]';
	arrDatenpunkt_Values_Pump[iDatapoints_Pump]:=LREAL_TO_FMTSTR(stPumpInformation.nSel_Setpoint_abs,2,TRUE);
	iDatapoints_Pump:=iDatapoints_Pump+1;
	
	arrDatenpunkt_IDs_Pump[iDatapoints_Pump]:='iPumpType	[]';
	arrDatenpunkt_Values_Pump[iDatapoints_Pump]:=UINT_TO_STRING(stPumpInformation.iPumpType);
	iDatapoints_Pump:=iDatapoints_Pump+1;
	
	arrDatenpunkt_IDs_Pump[iDatapoints_Pump]:='nMaxValue	[rpm, mWs]';
	arrDatenpunkt_Values_Pump[iDatapoints_Pump]:=LREAL_TO_FMTSTR(stPumpInformation.nMaxValue,0,TRUE);
	iDatapoints_Pump:=iDatapoints_Pump+1;
	
	arrDatenpunkt_IDs_Pump[iDatapoints_Pump]:='nMinValue	[rpm, mWs]';
	arrDatenpunkt_Values_Pump[iDatapoints_Pump]:=LREAL_TO_FMTSTR(stPumpInformation.nMinValue,0,TRUE);
	iDatapoints_Pump:=iDatapoints_Pump+1;

	arrDatenpunkt_IDs_Pump[iDatapoints_Pump]:='iCurrentWarning	[]';
	arrDatenpunkt_Values_Pump[iDatapoints_Pump]:=USINT_TO_STRING(stPumpInformation.iCurrentWarning);
	iDatapoints_Pump:=iDatapoints_Pump+1;

IF bReadOnly THEN	
	arrDatenpunkt_IDs_Pump[iDatapoints_Pump]:='';
	arrDatenpunkt_Values_Pump[iDatapoints_Pump]:='';
	iDatapoints_Pump:=iDatapoints_Pump+1;

	arrDatenpunkt_IDs_Pump[iDatapoints_Pump]:='';
	arrDatenpunkt_Values_Pump[iDatapoints_Pump]:='';
	iDatapoints_Pump:=iDatapoints_Pump+1;
	
	arrDatenpunkt_IDs_Pump[iDatapoints_Pump]:='';
	arrDatenpunkt_Values_Pump[iDatapoints_Pump]:='';
	iDatapoints_Pump:=iDatapoints_Pump-2;
	
ELSE
	arrDatenpunkt_IDs_Pump[iDatapoints_Pump]:='eBusCommand	[]';
	arrDatenpunkt_Values_Pump[iDatapoints_Pump]:=INT_TO_STRING(stPumpInformation.eBusCommand);
	iDatapoints_Pump:=iDatapoints_Pump+1;

	arrDatenpunkt_IDs_Pump[iDatapoints_Pump]:='eBusControlMode	[]';
	arrDatenpunkt_Values_Pump[iDatapoints_Pump]:=INT_TO_STRING(stPumpInformation.eBusControlMode);
	iDatapoints_Pump:=iDatapoints_Pump+1;
	
	arrDatenpunkt_IDs_Pump[iDatapoints_Pump]:='nBusSetpoint	[%, rpm, mWs]';
	arrDatenpunkt_Values_Pump[iDatapoints_Pump]:=LREAL_TO_FMTSTR(stPumpInformation.nBusSetpoint,2,TRUE);
	iDatapoints_Pump:=iDatapoints_Pump+1;
END_IF

END_FUNCTION_BLOCK

// Functions/SCALE
FUNCTION SCALE : LREAL
VAR_INPUT
	unscaledValue: LREAL;
	ScaleNum: REAL;
	ScaleDenum: REAL;
	ScaleOffset: REAL;
END_VAR

IF ScaleDenum <> 0 THEN
	SCALE:=ScaleNum/ScaleDenum*unscaledValue+ScaleOffset;
ELSE
	SCALE:=0;
END_IF

END_FUNCTION

// CAN/FB_SDO_WRITE
FUNCTION_BLOCK FB_SDO_WRITE
VAR_INPUT
	/// The AMSNetID addres of EL6751
	ADSNetID: STRING(23);
	/// The Port No. addresses the CANopen Node (see System Manager) 
	PortNr: WORD;
	/// This is the Index of the CANopen Object Dictionary Entry
	CO_Index: DWORD;
	/// This is the Sub-Index of the CANopen Object Dictionary Entry
	CO_SubIndex: DWORD;
	/// This is the Length of the CANopen Object Dictionary Entry
	DataLength: DWORD;
	/// only reset to FALSE after WriteDataFinished=TRUE
	StartWriting: BOOL;
	///This array contains the data to be written to the CANopen Object Dictionary
	WriteData: ARRAY[0..255] OF BYTE;
END_VAR
VAR_OUTPUT
	WriteDataFinished: BOOL;
	Error: DWORD;
END_VAR
VAR
	state: BYTE := 0;
	ADSWRITE: ADSWRITE;
END_VAR

CASE state OF
0:
	IF StartWriting THEN
		WriteDataFinished := FALSE;
		Error := 0;
		ADSWrite(
			NETID:= ADSNetID,
			PORT:= PortNr,
			IDXGRP:= CO_Index,
			IDXOFFS:= CO_SubIndex,
			LEN:= DataLength,
			SRCADDR:= ADR(WriteData),
			WRITE:= TRUE,
			TMOUT := T#1s
		);
		IF ADSWrite.err THEN
			state := 2;
			(*WriteDataFinished := TRUE;*)
			Error := ADSWrite.ErrId;
		ELSE
			state := 1;
		END_IF
	ELSE
		ADSWrite(
			NETID:= '',
			PORT:= PortNr,
			IDXGRP:= CO_Index,
			IDXOFFS:= CO_SubIndex,
			LEN:= DataLength,
			SRCADDR:= ADR(WriteData),
			WRITE:= FALSE,
			TMOUT := T#1s
		);
	END_IF

1:
	ADSWrite(WRITE:= FALSE);
	IF ADSWrite.err THEN
		state := 2;
		(*WriteDataFinished := TRUE;*)
		Error := ADSWrite.ErrId;
	ELSE
		IF NOT ADSWrite.busy THEN
			state := 2;
			(*WriteDataFinished := TRUE;*)
		END_IF
	END_IF

2:
	ADSWrite(WRITE:= FALSE);
	state := 0;
	WriteDataFinished := TRUE;
END_CASE

END_FUNCTION_BLOCK

// CAN/FB_SDO_READ
FUNCTION_BLOCK FB_SDO_READ
VAR_INPUT
	/// The AMSNetID addres of EL6751
	ADSNetID: STRING(23);
	/// This Port No. addresses the CANopen Node (see System Manager) 
	PortNr: WORD;
	/// This is the Index of the CANopen Object Dictionary Entry
	CO_Index: DWORD;
	/// This is the Sub-Index of the CANopen Object Dictionary Entry
	CO_SubIndex: DWORD;
	/// This is the Length of the CANopen Object Dictionary Entry
	DataLength: DWORD;
	/// only reset to FALSE after ReadDataAvailable=TRUE
	StartReading: BOOL;
END_VAR
VAR_OUTPUT
	ReadData: ARRAY[0..255] OF BYTE;
	ReadDataAvailable: BOOL;
	Error: DWORD;
END_VAR
VAR
	state: BYTE := 0;
	ADSREAD: ADSREAD;
END_VAR

CASE state OF
0:
	IF StartReading THEN
		ReadDataAvailable := FALSE;
		Error := 0;
		ADSRead(
			NETID:= ADSNetID,
			PORT:= PortNr,
			IDXGRP:= CO_Index,
			IDXOFFS:= CO_SubIndex,
			LEN:= DataLength,
			DESTADDR:= ADR(ReadData),
			READ:= TRUE,
			TMOUT := T#1s
		);
		IF ADSRead.err THEN
			state := 2;
			(*ReadDataAvailable := TRUE;*)
			Error := ADSRead.ErrId;
		ELSE
			state := 1;
		END_IF
	ELSE
		ADSRead(
			NETID:= ADSNetID,
			PORT:= PortNr,
			IDXGRP:= CO_Index,
			IDXOFFS:= CO_SubIndex,
			LEN:= DataLength,
			DESTADDR:= ADR(ReadData),
			READ:= FALSE,
			TMOUT := T#1s
		);
	END_IF

1:
	ADSRead(READ:= FALSE);
	IF ADSRead.err THEN
		state := 2;
		(*ReadDataAvailable := TRUE;*)
		Error := ADSRead.ErrId;
	ELSE
		IF NOT ADSRead.busy THEN
			state := 2;
			(*ReadDataAvailable := TRUE;*)
		END_IF
	END_IF

2: 
	ADSRead(READ:= FALSE);
	ReadDataAvailable := TRUE;
	state := 0;
END_CASE

END_FUNCTION_BLOCK

// CAN/StratosGiga_IPE/FB_StratosGIGA_IPE
FUNCTION_BLOCK FB_StratosGIGA_IPE
VAR_INPUT
	// CAN configuration
		sCAN_NetID								:STRING (23);	// NetID of CAN Master
		iCAN_NodeID								:UINT;		// NodeId (automatic calculation of Port No.
	// control configuration
		bReadOnly								:BOOL;		// deactivate pump control
		bUseAbsoluteSetpoint					:BOOL;		// use rpm or mWs instead of %
		bExternalCommandOverride				:BOOL:=TRUE;	// Use  for pump control Struct instead of PumpInformationStruct to control the pump
		stPumpControl							:StratosControl; // Struct for control pump by external PLC Code

END_VAR
VAR_OUTPUT
	// Error
		iReadError								:UINT;	// number of Errors (read)
		iWriteError								:UINT;	// number of Errors (write)
	
	// Structure	
		stPumpInformation						:WILO_StratosGiga_IPE; // Information (Control) of pump
			
	// Logging
		arrDatenpunkt_IDs_Pump					:ARRAY [0..99] OF T_MaxString;			(*Beschreibung der Datenpunkte*)
		arrDatenpunkt_Values_Pump				:ARRAY [0..99] OF T_MaxString;			(*Messwerte der Datenpunkte*)
		iDatapoints_Pump						:INT			:=0;
END_VAR
VAR	
	// Datapoints
(*		iSpeed									:UINT;			//[rpm]	
		nPressure								:LREAL;			//[mWs]
		nFlow									:LREAL;			//[m³/h]		
		nInputPower								:LREAL;			//[W]
		nConsumption							:LREAL;			//[kWh]	
		nMediumTemp								:LREAL;			//[°C]
		nOperatingHours							:LREAL;			//[h]		
		eEff_Command							:eEffCommand;	
		eEff_ControlMode						:eBusControlMode;	
		nEff_Setpoint							:LREAL;			//[%]
		nEff_Setpoint_abs						:LREAL;			//[rpm, mWs]
		eSel_Command							:eEffCommand;
		eSel_ControlMode						:eBusControlMode;
		nSel_Setpoint							:LREAL;			//[%]
		nSel_Setpoint_abs						:LREAL;			//[rpm, mWs]
		iPumpType								:UINT;			//[PumpType]	
		nMaxValue								:LREAL;			//[mWs], [rpm]
		iCurrentWarning							:USINT;			//[Error Code]		
*)
	// Read
		imaxValue								:UINT;	
		iInputPower								:UDINT;	
		iPressure								:UINT;			
		iFlow									:UINT;	
		ieff_Setpoint							:INT;					
		iEff_ControlMode					 	:USINT;
		ieff_Command							:USINT;	
		iSel_Setpoint							:INT;					
		iSel_ControlMode					 	:USINT;
		iSel_Command							:USINT;
		iConsumption							:UDINT;	
		iOperatingHours							:UDINT;
		iBusStatus								:USINT;
		iControlStatus 							:USINT;
		iReadyForOperation 						:USINT;
		iPumpIsOperating 						:USINT;
		iServiceRequired 						:USINT;
		iElectricalCurrent 						:UDINT;
		iVoltageLevel 							:UINT;
		iCalculatedPressure 					:UINT;
		iWindingTemperature 					:UINT;
		iModuleTemperature 						:UINT;
		iElectronicTemperature 					:UINT;
		iCalculatedTorque 						:UINT;
		iSpecialStatus 							:USINT;
		iInternalSetpoint 						:UINT;
		iSpeedObserved 							:UINT;
		iCharacteristicCurveIndex 				:USINT;
		iMotorNumber 							:USINT;
		iCalculatedPressureCorrected 			:UINT;
		iSperrzeitDPspitzenlast 				:USINT;
		iE255Index 								:UINT;
		iE255Value 								:USINT;
		iFUlimits 								:USINT;		
		

	// Write
		iBusCommand								:USINT;			//16#61=PumpOn; 16#60=PumpOff
		iBusControlMode					 		:USINT;			//0=nc; 5=dpc; 6=dpv
		iBusSetpoint					 		:INT;			
	
	// CAN
		State_CAN								:INT		:=0;	
	
	// CAN-ini
		CAN_NodePort							:WORD;
		
	// CAN-Datenpunkteigenschaften
		CAN_Index								:DWORD;
		CAN_Subindex							:DWORD;
		CAN_Length								:DWORD;
		CAN_RW_Mode								:INT		:=0;
		CAN_Start								:BOOL		:=FALSE;
		iDpAddres								:POINTER TO ARRAY [0..7] OF BYTE;
		bReadSuccesfull							:BOOL;
		
	// CAN-SDO_Write Baustein
		CAN_SDO_WRITE							:FB_SDO_WRITE;
		CAN_WriteData							:ARRAY[0..255] OF BYTE;
		CAN_WriteError							:DWORD;
		
	// CAN-SDO_Read Baustein
		CAN_SDO_READ							:FB_SDO_READ;
		CAN_ReadData							:ARRAY[0..255] OF BYTE;
		CAN_ReadError							:DWORD;
		CAN_ScaleNum							:REAL			:=1;
		CAN_ScaleDenum							:REAL			:=1;
		CAN_ScaleOffset							:REAL			:=0;	
		CAN_Description							:STRING;
		CAN_Datatype							:Datatyp;
		CAN_Unit								:STRING;
		CAN_Unit_abs							:STRING;
END_VAR

// calculate NodePort by NodeID
CAN_NodePort:=16#1000+iCAN_NodeID;	

IF bExternalCommandOverride THEN
	stPumpInformation.eBusCommand:= stPumpControl.eBusCommand;
	stPumpInformation.eBusControlMode:= stPumpControl.eBusControlMode;
	stPumpInformation.nBusSetpoint:= stPumpControl.nBusSetpoint;
END_IF

// SDO-Pumpendatenpunkte	
	CASE State_CAN OF
	0:  // Initialisierung
		State_CAN := 1;
		
	1:	// Datenpunkt Pump Type
		CAN_Index:=16#2182;
		CAN_Subindex:=16#1;
		CAN_Length:=16#2;
		CAN_RW_Mode:=1;
		CAN_ScaleNum:=1;
		CAN_ScaleDenum:=1;
		CAN_ScaleOffset:=0;
		CAN_Description:='PumpType';
		CAN_Unit:='-';
		CAN_Datatype:=9;
		iDpAddres:=ADR(stPumpInformation.iPumpType);
		
		IF bReadSuccesfull THEN
			stPumpinformation.arrPumpInformation[State_CAN].sValue:=UINT_TO_STRING(stPumpInformation.iPumpType);
			bReadSuccesfull:=FALSE;
			State_CAN := State_CAN+1;
		END_IF
		
	2:	// Datenpunkt maxFörderhöhe [mWs] bzw. maxDrehzahl [rpm]
		CASE ieff_ControlMode OF
			0:		CAN_Index:=16#21A1;
					CAN_ScaleNum:=1;
					CAN_ScaleDenum:=1;
					CAN_ScaleOffset:=0;
					CAN_Unit:='rpm';
					CAN_Unit_abs:='rpm';
					
			5:		CAN_Index:=16#21AD;
					CAN_ScaleNum:=102;
					CAN_ScaleDenum:=10000;
					CAN_ScaleOffset:=0;
					CAN_Unit:='mWs';
					CAN_Unit_abs:='mWs';
			
			6:		CAN_Index:=16#21A5;
					CAN_ScaleNum:=102;
					CAN_ScaleDenum:=10000;
					CAN_ScaleOffset:=0;
					CAN_Unit:='mWs';
					CAN_Unit_abs:='mWs';
			
			ELSE	CAN_Index:=16#21AD;
					CAN_ScaleNum:=102;
					CAN_ScaleDenum:=10000;
					CAN_ScaleOffset:=0;
					CAN_Unit:='mWs';	
					CAN_Unit_abs:='mWs';	
		END_CASE
		
		CAN_Subindex:=16#0;
		CAN_Length:=16#2;	
		CAN_RW_Mode:=1;
		CAN_Description:='maxValue';
		CAN_Datatype:=13;
		iDpAddres:=ADR(imaxValue);
		
		IF bReadSuccesfull THEN
			stPumpInformation.nmaxValue:=SCALE(imaxValue,CAN_ScaleNum,CAN_ScaleDenum,CAN_ScaleOffset);			
			stPumpinformation.arrPumpInformation[State_CAN].sValue:=LREAL_TO_STRING(stPumpInformation.nMaxValue);
			bReadSuccesfull:=FALSE;			
			State_CAN := State_CAN+1;
		END_IF

	3:	// Datenpunkt Speed [rpm]
		CAN_Index:=16#2083;
		CAN_Subindex:=16#1;
		CAN_Length:=16#2;
		CAN_RW_Mode:=1;
		CAN_ScaleNum:=1;
		CAN_ScaleDenum:=1;
		CAN_ScaleOffset:=0;
		CAN_Description:='Speed';
		CAN_Unit:='rpm';
		CAN_Datatype:=9;
		iDpAddres:=ADR(stPumpInformation.ispeed);
		
		IF bReadSuccesfull THEN
			stPumpinformation.arrPumpInformation[State_CAN].sValue:=UINT_TO_STRING(stPumpInformation.ispeed);
			bReadSuccesfull:=FALSE;	
			State_CAN := State_CAN+1;
		END_IF
		
	4:	// Datenpunkt Flow [m^3/h]
		CAN_Index:=16#2087;
		CAN_Subindex:=16#0;
		CAN_Length:=16#2;
		CAN_RW_Mode:=1;
		CAN_ScaleNum:=1;
		CAN_ScaleDenum:=10;
		CAN_ScaleOffset:=0;
		CAN_Description:='EstimatedFlow';
		CAN_Unit:='m³/h';
		CAN_Datatype:=13;
		iDpAddres:=ADR(iflow);
		
		IF bReadSuccesfull THEN
			IF iFlow >= 65534 THEN
				stPumpInformation.nflow:=-99999;
				stPumpinformation.arrPumpInformation[State_CAN].sValue:='naN';	
			ELSE
				stPumpInformation.nflow:=SCALE(iflow,CAN_ScaleNum,CAN_ScaleDenum,CAN_ScaleOffset);
				stPumpinformation.arrPumpInformation[State_CAN].sValue:=LREAL_TO_STRING(stPumpInformation.nflow);				
			END_IF
			bReadSuccesfull:=FALSE;	
			State_CAN := State_CAN+1;
		END_IF
			
	5:	// Datenpunkt Consumption [kWh]
		CAN_Index:=16#2113;
		CAN_Subindex:=16#0;
		CAN_Length:=16#4;
		CAN_RW_Mode:=1;
		CAN_ScaleNum:=1;
		CAN_ScaleDenum:=10;
		CAN_ScaleOffset:=0;
		CAN_Description:='Consumption';
		CAN_Unit:='kWh';
		CAN_Datatype:=13;
		iDpAddres:=ADR(iConsumption);
		
		IF bReadSuccesfull THEN
			stPumpInformation.nConsumption:=SCALE(iConsumption,CAN_ScaleNum,CAN_ScaleDenum,CAN_ScaleOffset);
			stPumpinformation.arrPumpInformation[State_CAN].sValue:=LREAL_TO_STRING(stPumpInformation.nConsumption);
			bReadSuccesfull:=FALSE;	
			State_CAN := State_CAN+1;		
		END_IF
	
	6:	// Datenpunkt Operating Hours [h]
		CAN_Index:=16#2101;
		CAN_Subindex:=16#0;
		CAN_Length:=16#4;
		CAN_RW_Mode:=1;
		CAN_ScaleNum:=1;
		CAN_ScaleDenum:=60;
		CAN_ScaleOffset:=0;
		CAN_Description:='OperationTimeResettable';
		CAN_Unit:='kWh';
		CAN_Datatype:=13;
		iDpAddres:=ADR(iOperatingHours);
		
		IF bReadSuccesfull THEN
			stPumpInformation.nOperatingHours:=SCALE(iOperatingHours,CAN_ScaleNum,CAN_ScaleDenum,CAN_ScaleOffset);			
			stPumpinformation.arrPumpInformation[State_CAN].sValue:=LREAL_TO_STRING(stPumpInformation.nOperatingHours);
			bReadSuccesfull:=FALSE;	
			State_CAN := State_CAN+1;
		END_IF
		
	7:	// Datenpunkt Current Warning
		CAN_Index:=16#20C1;
		CAN_Subindex:=16#0;
		CAN_Length:=16#1;
		CAN_RW_Mode:=1;
		CAN_ScaleNum:=1;
		CAN_ScaleDenum:=1;
		CAN_ScaleOffset:=0;
		CAN_Description:='CurrentWarning_Error';
		CAN_Unit:='-';
		CAN_Datatype:=8;
		iDpAddres:=ADR(stPumpInformation.iCurrentWarning);
		
		IF bReadSuccesfull THEN
			stPumpinformation.arrPumpInformation[State_CAN].sValue:=USINT_TO_STRING(stPumpInformation.iCurrentWarning);
			bReadSuccesfull:=FALSE;	
			State_CAN := State_CAN+1;
		END_IF
		
	8: 	// Datenpunkt Input Power
		CAN_Index:=16#2090;
		CAN_Subindex:=16#0;
		CAN_Length:=16#4;
		CAN_RW_Mode:=1;
		CAN_ScaleNum:=1;
		CAN_ScaleDenum:=1000;
		CAN_ScaleOffset:=0;
		CAN_Description:='InputPower';
		CAN_Unit:='W';
		CAN_Datatype:=13;
		iDpAddres:=ADR(iInputPower);
		
		IF bReadSuccesfull THEN
			stPumpInformation.nInputPower:=SCALE(iInputPower,CAN_ScaleNum,CAN_ScaleDenum,CAN_ScaleOffset);
			stPumpinformation.arrPumpInformation[State_CAN].sValue:=LREAL_TO_STRING(stPumpInformation.nInputPower);
			bReadSuccesfull:=FALSE;	
			State_CAN := State_CAN+1;
		END_IF
		
	9: 	// Datenpunkt Pressure
		CAN_Index:=16#208A;
		CAN_Subindex:=16#0;
		CAN_Length:=16#2;
		CAN_RW_Mode:=1;
		CAN_ScaleNum:=102;
		CAN_ScaleDenum:=10000;
		CAN_ScaleOffset:=0;
		CAN_Description:='Pressure';
		CAN_Unit:='mWs';
		CAN_Datatype:=13;
		iDpAddres:=ADR(iPressure);
		
		IF bReadSuccesfull THEN
			IF iPressure >= 65534 THEN
				stPumpInformation.nPressure:=-99999;
				stPumpinformation.arrPumpInformation[State_CAN].sValue:='naN';	
			ELSE
				stPumpInformation.nPressure:=SCALE(iPressure,CAN_ScaleNum,CAN_ScaleDenum,CAN_ScaleOffset);
				stPumpinformation.arrPumpInformation[State_CAN].sValue:=LREAL_TO_STRING(stPumpInformation.nPressure);	
			END_IF	

			bReadSuccesfull:=FALSE;	
			State_CAN := State_CAN+1;
		END_IF
		
	10: // Actual Value Sensor Source
		CAN_Index:=16#2077;
		CAN_Subindex:=16#0;
		CAN_Length:=16#1;
		CAN_RW_Mode:=1;
		CAN_ScaleNum:=1;
		CAN_ScaleDenum:=1;
		CAN_ScaleOffset:=0;
		CAN_Description:='ActualValueSensorSource';
		CAN_Unit:='-';
		CAN_Datatype:=8;
		iDpAddres:=ADR(stPumpInformation.iPressureSensorSource);
		
		IF bReadSuccesfull THEN
			stPumpinformation.arrPumpInformation[State_CAN].sValue:=USINT_TO_STRING(stPumpInformation.iPressureSensorSource);
			bReadSuccesfull:=FALSE;	
			State_CAN := State_CAN+1;
		END_IF
		
	11: // Datenpunkt effective Capacity
		CAN_Index:=16#2040;
		CAN_Subindex:=16#0;
		CAN_Length:=16#2;
		CAN_RW_Mode:=1;
		CAN_ScaleNum:=1;
		CAN_ScaleDenum:=100;
		CAN_ScaleOffset:=0;
		CAN_Description:='EffectiveCapacity';
		CAN_Unit:='%';
		CAN_Datatype:=13;
		iDpAddres:=ADR(ieff_Setpoint);
		
		IF bReadSuccesfull THEN
			stPumpInformation.neff_Setpoint:=SCALE(ieff_Setpoint,CAN_ScaleNum,CAN_ScaleDenum,CAN_ScaleOffset);
			stPumpInformation.neff_Setpoint_abs:=stPumpInformation.neff_Setpoint/100*stPumpInformation.nMaxValue;
			IF bUseAbsoluteSetpoint THEN
				stPumpinformation.arrPumpInformation[State_CAN].sValue:=LREAL_TO_STRING(stPumpInformation.neff_Setpoint_abs);
				stPumpinformation.arrPumpInformation[State_CAN].sUnit:=CAN_Unit_abs;	
			ELSE
				stPumpinformation.arrPumpInformation[State_CAN].sValue:=LREAL_TO_STRING(stPumpInformation.neff_Setpoint);
			END_IF
			bReadSuccesfull:=FALSE;	
			State_CAN := State_CAN+1;
		END_IF
				
	12: // Datenpunkt effective Control Mode
		CAN_Index:=16#2041;
		CAN_Subindex:=16#0;
		CAN_Length:=16#1;
		CAN_RW_Mode:=1;
		CAN_ScaleNum:=1;
		CAN_ScaleDenum:=1;
		CAN_ScaleOffset:=0;
		CAN_Description:='EffectiveControlMode';
		CAN_Unit:='-';
		CAN_Datatype:=15;
		iDpAddres:=ADR(ieff_ControlMode);
		
		IF bReadSuccesfull THEN
			stPumpInformation.eeff_ControlMode:=USINT_TO_INT(ieff_ControlMode);
			stPumpinformation.arrPumpInformation[State_CAN].sValue:=USINT_TO_STRING(ieff_ControlMode);
			bReadSuccesfull:=FALSE;	
			State_CAN := State_CAN+1;
		END_IF

	13: // Datenpunkt effective Command
		CAN_Index:=16#2042;
		CAN_Subindex:=16#0;
		CAN_Length:=16#1;
		CAN_RW_Mode:=1;
		CAN_ScaleNum:=1;
		CAN_ScaleDenum:=1;
		CAN_ScaleOffset:=0;
		CAN_Description:='EffectiveCommand';
		CAN_Unit:='-';
		CAN_Datatype:=15;
		iDpAddres:=ADR(ieff_Command);
		
		IF bReadSuccesfull THEN
			stPumpInformation.eeff_Command:=USINT_TO_INT(ieff_Command);
			stPumpinformation.arrPumpInformation[State_CAN].sValue:=USINT_TO_STRING(ieff_Command);
			bReadSuccesfull:=FALSE;	
			State_CAN := State_CAN+1;
		END_IF

	14: // Datenpunkt Selected BusSetpoint
		CAN_Index:=16#2048;
		CAN_Subindex:=16#0;
		CAN_Length:=16#2;
		CAN_RW_Mode:=1;
		CAN_ScaleNum:=1;
		CAN_ScaleDenum:=100;
		CAN_ScaleOffset:=0;
		CAN_Description:='SelectedSetpoint';
		CAN_Unit:='%';
		CAN_Datatype:=13;
		iDpAddres:=ADR(iSel_Setpoint);
		
		IF bReadSuccesfull THEN
			stPumpInformation.nSel_Setpoint:=SCALE(iSel_Setpoint,CAN_ScaleNum,CAN_ScaleDenum,CAN_ScaleOffset);
			stPumpInformation.nSel_Setpoint_abs:=stPumpInformation.nSel_Setpoint/100*stPumpInformation.nMaxValue;
			IF bUseAbsoluteSetpoint THEN
				stPumpinformation.arrPumpInformation[State_CAN].sValue:=LREAL_TO_STRING(stPumpInformation.nSel_Setpoint_abs);
				stPumpinformation.arrPumpInformation[State_CAN].sUnit:=CAN_Unit_abs;	
			ELSE
				stPumpinformation.arrPumpInformation[State_CAN].sValue:=LREAL_TO_STRING(stPumpInformation.nSel_Setpoint);
			END_IF		
			bReadSuccesfull:=FALSE;	
			State_CAN := State_CAN+1;
		END_IF
		
	15:	// Datenpunkt Selected Control Mode
		CAN_Index:=16#2049;
		CAN_Subindex:=16#0;
		CAN_Length:=16#1;
		CAN_RW_Mode:=1;
		CAN_ScaleNum:=1;
		CAN_ScaleDenum:=1;
		CAN_ScaleOffset:=0;
		CAN_Description:='SelectedControlMode';
		CAN_Unit:='-';
		CAN_Datatype:=15;
		iDpAddres:=ADR(iSel_ControlMode);
		
		IF bReadSuccesfull THEN
			stPumpInformation.eSel_ControlMode:=USINT_TO_INT(iSel_ControlMode);
			stPumpinformation.arrPumpInformation[State_CAN].sValue:=USINT_TO_STRING(iSel_ControlMode);
			bReadSuccesfull:=FALSE;	
			State_CAN := State_CAN+1;
		END_IF
		
	16:	// Datenpunkt Selected BusCommand
		CAN_Index:=16#204A;
		CAN_Subindex:=16#0;
		CAN_Length:=16#1;
		CAN_RW_Mode:=1;
		CAN_ScaleNum:=1;
		CAN_ScaleDenum:=1;
		CAN_ScaleOffset:=0;
		CAN_Description:='SelectedCommand';
		CAN_Unit:='-';
		CAN_Datatype:=15;
		iDpAddres:=ADR(iSel_Command);
		
		IF bReadSuccesfull THEN
			stPumpInformation.eSel_Command:=USINT_TO_INT(iSel_Command);
			stPumpinformation.arrPumpInformation[State_CAN].sValue:=USINT_TO_STRING(iSel_Command);
			bReadSuccesfull:=FALSE;	
			State_CAN := State_CAN+1;
		END_IF

	17:	// Datenpunkt BusStatus
		CAN_Index:=16#2054;
		CAN_Subindex:=16#0;
		CAN_Length:=16#1;
		CAN_RW_Mode:=1;
		CAN_ScaleNum:=1;
		CAN_ScaleDenum:=1;
		CAN_ScaleOffset:=0;
		CAN_Description:='BusStatus';
		CAN_Unit:='-';
		CAN_Datatype:=8;
		iDpAddres:=ADR(iBusStatus);
		
		IF bReadSuccesfull THEN
			stPumpInformation.iBusStatus:=iBusStatus;
			stPumpinformation.arrPumpInformation[State_CAN].sValue:=USINT_TO_STRING(iBusStatus);
			bReadSuccesfull:=FALSE;	
			State_CAN := State_CAN+1;
		END_IF
		
	18:	// Datenpunkt ControlStatus
		CAN_Index:=16#2056;
		CAN_Subindex:=16#0;
		CAN_Length:=16#1;
		CAN_RW_Mode:=1;
		CAN_ScaleNum:=1;
		CAN_ScaleDenum:=1;
		CAN_ScaleOffset:=0;
		CAN_Description:='ControlStatus';
		CAN_Unit:='-';
		CAN_Datatype:=8;
		iDpAddres:=ADR(iControlStatus);
		
		IF bReadSuccesfull THEN
			stPumpInformation.iControlStatus:=iControlStatus;
			stPumpinformation.arrPumpInformation[State_CAN].sValue:=USINT_TO_STRING(iControlStatus);
			bReadSuccesfull:=FALSE;	
			State_CAN := State_CAN+1;
		END_IF
		
	19:	// Datenpunkt ReadyForOperation
		CAN_Index:=16#2058;
		CAN_Subindex:=16#0;
		CAN_Length:=16#1;
		CAN_RW_Mode:=1;
		CAN_ScaleNum:=1;
		CAN_ScaleDenum:=1;
		CAN_ScaleOffset:=0;
		CAN_Description:='ReadyForOperation';
		CAN_Unit:='-';
		CAN_Datatype:=8;
		iDpAddres:=ADR(iReadyForOperation);
		
		IF bReadSuccesfull THEN
			stPumpInformation.iReadyForOperation:=iReadyForOperation;
			stPumpinformation.arrPumpInformation[State_CAN].sValue:=USINT_TO_STRING(iReadyForOperation);
			bReadSuccesfull:=FALSE;	
			State_CAN := State_CAN+1;
		END_IF
		
	20:	// Datenpunkt PumpIsOperating
		CAN_Index:=16#205A;
		CAN_Subindex:=16#0;
		CAN_Length:=16#1;
		CAN_RW_Mode:=1;
		CAN_ScaleNum:=1;
		CAN_ScaleDenum:=1;
		CAN_ScaleOffset:=0;
		CAN_Description:='PumpIsOperating';
		CAN_Unit:='-';
		CAN_Datatype:=8;
		iDpAddres:=ADR(iPumpIsOperating);
		
		IF bReadSuccesfull THEN
			stPumpInformation.iPumpIsOperating:=iPumpIsOperating;
			stPumpinformation.arrPumpInformation[State_CAN].sValue:=USINT_TO_STRING(iPumpIsOperating);
			bReadSuccesfull:=FALSE;	
			State_CAN := State_CAN+1;
		END_IF
		
	21:	// Datenpunkt ServiceRequired
		CAN_Index:=16#205C;
		CAN_Subindex:=16#0;
		CAN_Length:=16#1;
		CAN_RW_Mode:=1;
		CAN_ScaleNum:=1;
		CAN_ScaleDenum:=1;
		CAN_ScaleOffset:=0;
		CAN_Description:='ServiceRequired';
		CAN_Unit:='-';
		CAN_Datatype:=8;
		iDpAddres:=ADR(iServiceRequired);
		
		IF bReadSuccesfull THEN
			stPumpInformation.iServiceRequired:=iServiceRequired;
			stPumpinformation.arrPumpInformation[State_CAN].sValue:=USINT_TO_STRING(iServiceRequired);
			bReadSuccesfull:=FALSE;	
			State_CAN := State_CAN+1;
		END_IF
		
	22: 	// Datenpunkt ElectricalCurrent
		CAN_Index:=16#2091;
		CAN_Subindex:=16#0;
		CAN_Length:=16#4;
		CAN_RW_Mode:=1;
		CAN_ScaleNum:=1;
		CAN_ScaleDenum:=1000;
		CAN_ScaleOffset:=0;
		CAN_Description:='ElectricalCurrent';
		CAN_Unit:='A';
		CAN_Datatype:=13;
		iDpAddres:=ADR(iElectricalCurrent);
		
		IF bReadSuccesfull THEN
			stPumpInformation.nElectricalCurrent:=SCALE(iElectricalCurrent,CAN_ScaleNum,CAN_ScaleDenum,CAN_ScaleOffset);
			stPumpinformation.arrPumpInformation[State_CAN].sValue:=LREAL_TO_STRING(stPumpInformation.nElectricalCurrent);
			bReadSuccesfull:=FALSE;	
			State_CAN := State_CAN+1;
		END_IF
		
		
	23: 	// Datenpunkt VoltageLevel
		CAN_Index:=16#2092;
		CAN_Subindex:=16#1;
		CAN_Length:=16#2;
		CAN_RW_Mode:=1;
		CAN_ScaleNum:=1;
		CAN_ScaleDenum:=1;
		CAN_ScaleOffset:=0;
		CAN_Description:='VoltageLevel';
		CAN_Unit:='V';
		CAN_Datatype:=13;
		iDpAddres:=ADR(iVoltageLevel);
		
		IF bReadSuccesfull THEN
			stPumpInformation.nVoltageLevel:=SCALE(iVoltageLevel,CAN_ScaleNum,CAN_ScaleDenum,CAN_ScaleOffset);
			stPumpinformation.arrPumpInformation[State_CAN].sValue:=LREAL_TO_STRING(stPumpInformation.nVoltageLevel);
			bReadSuccesfull:=FALSE;	
			State_CAN := State_CAN+1;
		END_IF	
		
	24: 	
		CAN_RW_Mode:=0;
		State_CAN := 39;	// jump to case 39, other dp only in developer mode	
(*
	24: 	// Datenpunkt CalculatedPressure
		CAN_Index:=16#26C0;
		CAN_Subindex:=16#0;
		CAN_Length:=16#2;
		CAN_RW_Mode:=1;
		CAN_ScaleNum:=1;
		CAN_ScaleDenum:=10;
		CAN_ScaleOffset:=0;
		CAN_Description:='CalculatedPressure';
		CAN_Unit:='mWs';
		CAN_Datatype:=13;
		iDpAddres:=ADR(iCalculatedPressure);
		
		IF bReadSuccesfull THEN
			stPumpInformation.nCalculatedPressure:=SCALE(iCalculatedPressure,CAN_ScaleNum,CAN_ScaleDenum,CAN_ScaleOffset);
			stPumpinformation.arrPumpInformation[State_CAN].sValue:=LREAL_TO_STRING(stPumpInformation.nCalculatedPressure);
			bReadSuccesfull:=FALSE;	
			State_CAN := State_CAN+1;
		END_IF	

	25:	// Datenpunkt WindingTemperature
		CAN_Index:=16#206C1;
		CAN_Subindex:=16#0;
		CAN_Length:=16#2;
		CAN_RW_Mode:=1;
		CAN_ScaleNum:=1;
		CAN_ScaleDenum:=1;
		CAN_ScaleOffset:=0;
		CAN_Description:='WindingTemperature';
		CAN_Unit:='ADC Value';
		CAN_Datatype:=9;
		iDpAddres:=ADR(iWindingTemperature);
		
		IF bReadSuccesfull THEN
			stPumpInformation.iWindingTemperature:=iWindingTemperature;
			stPumpinformation.arrPumpInformation[State_CAN].sValue:=UINT_TO_STRING(iWindingTemperature);
			bReadSuccesfull:=FALSE;	
			State_CAN := State_CAN+1;
		END_IF		
		
	26:	// Datenpunkt ModuleTemperature
		CAN_Index:=16#206C2;
		CAN_Subindex:=16#0;
		CAN_Length:=16#2;
		CAN_RW_Mode:=1;
		CAN_ScaleNum:=1;
		CAN_ScaleDenum:=1;
		CAN_ScaleOffset:=0;
		CAN_Description:='ModuleTemperature';
		CAN_Unit:='ADC Value';
		CAN_Datatype:=9;
		iDpAddres:=ADR(iModuleTemperature);
		
		IF bReadSuccesfull THEN
			stPumpInformation.iModuleTemperature:=iModuleTemperature;
			stPumpinformation.arrPumpInformation[State_CAN].sValue:=UINT_TO_STRING(iModuleTemperature);
			bReadSuccesfull:=FALSE;	
			State_CAN := State_CAN+1;
		END_IF			
		
	27:	// Datenpunkt ElectronicTemperature
		CAN_Index:=16#206C3;
		CAN_Subindex:=16#0;
		CAN_Length:=16#2;
		CAN_RW_Mode:=1;
		CAN_ScaleNum:=1;
		CAN_ScaleDenum:=1;
		CAN_ScaleOffset:=0;
		CAN_Description:='ElectronicTemperature';
		CAN_Unit:='ADC Value';
		CAN_Datatype:=9;
		iDpAddres:=ADR(iElectronicTemperature);
		
		IF bReadSuccesfull THEN
			stPumpInformation.iElectronicTemperature:=iElectronicTemperature;
			stPumpinformation.arrPumpInformation[State_CAN].sValue:=UINT_TO_STRING(iElectronicTemperature);
			bReadSuccesfull:=FALSE;	
			State_CAN := State_CAN+1;
		END_IF	

	28: // Datenpunkt CalculatedTorque
		CAN_Index:=16#26C4;
		CAN_Subindex:=16#1;
		CAN_Length:=16#2;
		CAN_RW_Mode:=1;
		CAN_ScaleNum:=1;
		CAN_ScaleDenum:=100;
		CAN_ScaleOffset:=0;
		CAN_Description:='CalculatedTorque';
		CAN_Unit:='Nm';
		CAN_Datatype:=13;
		iDpAddres:=ADR(iCalculatedTorque);
		
		IF bReadSuccesfull THEN
			stPumpInformation.nCalculatedTorque:=SCALE(iCalculatedTorque,CAN_ScaleNum,CAN_ScaleDenum,CAN_ScaleOffset);
			stPumpinformation.arrPumpInformation[State_CAN].sValue:=LREAL_TO_STRING(stPumpInformation.nCalculatedTorque);
			bReadSuccesfull:=FALSE;	
			State_CAN := State_CAN+1;
		END_IF	
		
	29:	// Datenpunkt SpecialStatus
		CAN_Index:=16#26C5;
		CAN_Subindex:=16#0;
		CAN_Length:=16#1;
		CAN_RW_Mode:=1;
		CAN_ScaleNum:=1;
		CAN_ScaleDenum:=1;
		CAN_ScaleOffset:=0;
		CAN_Description:='SpecialStatus';
		CAN_Unit:='-';
		CAN_Datatype:=8;
		iDpAddres:=ADR(iSpecialStatus);
		
		IF bReadSuccesfull THEN
			stPumpInformation.iSpecialStatus:=iSpecialStatus;
			stPumpinformation.arrPumpInformation[State_CAN].sValue:=USINT_TO_STRING(iSpecialStatus);
			bReadSuccesfull:=FALSE;	
			State_CAN := State_CAN+1;
		END_IF		
		
	30:	// Datenpunkt InternalSetpoint
		CAN_Index:=16#26C6;
		CAN_Subindex:=16#0;
		CAN_Length:=16#2;
		CAN_RW_Mode:=1;
		CAN_ScaleNum:=1;
		CAN_ScaleDenum:=10;
		CAN_ScaleOffset:=0;
		CAN_Description:='InternalSetpoint';
		CAN_Unit:='mWs';
		CAN_Datatype:=13;
		iDpAddres:=ADR(iInternalSetpoint);
		
		IF bReadSuccesfull THEN
			stPumpInformation.nInternalSetpoint:=SCALE(iInternalSetpoint,CAN_ScaleNum,CAN_ScaleDenum,CAN_ScaleOffset);
			stPumpinformation.arrPumpInformation[State_CAN].sValue:=LREAL_TO_STRING(stPumpInformation.nInternalSetpoint);
			bReadSuccesfull:=FALSE;	
			State_CAN := State_CAN+1;
		END_IF	
		
	31:	// Datenpunkt SpeedObserved
		CAN_Index:=16#26C7;
		CAN_Subindex:=16#0;
		CAN_Length:=16#2;
		CAN_RW_Mode:=1;
		CAN_ScaleNum:=1;
		CAN_ScaleDenum:=1;
		CAN_ScaleOffset:=0;
		CAN_Description:='SpeedObserved';
		CAN_Unit:='rpm';
		CAN_Datatype:=9;
		iDpAddres:=ADR(iSpeedObserved);
		
		IF bReadSuccesfull THEN
			stPumpInformation.iSpeedObserved:=iSpeedObserved;
			stPumpinformation.arrPumpInformation[State_CAN].sValue:=UINT_TO_STRING(iSpeedObserved);
			bReadSuccesfull:=FALSE;	
			State_CAN := State_CAN+1;
		END_IF	

	32:	// Datenpunkt CharacteristicCurveIndex
		CAN_Index:=16#26C8;
		CAN_Subindex:=16#0;
		CAN_Length:=16#1;
		CAN_RW_Mode:=1;
		CAN_ScaleNum:=1;
		CAN_ScaleDenum:=1;
		CAN_ScaleOffset:=0;
		CAN_Description:='CharacteristicCurveIndex';
		CAN_Unit:='-';
		CAN_Datatype:=8;
		iDpAddres:=ADR(iCharacteristicCurveIndex);
		
		IF bReadSuccesfull THEN
			stPumpInformation.iCharacteristicCurveIndex:=iCharacteristicCurveIndex;
			stPumpinformation.arrPumpInformation[State_CAN].sValue:=USINT_TO_STRING(iCharacteristicCurveIndex);
			bReadSuccesfull:=FALSE;	
			State_CAN := State_CAN+1;
		END_IF		

	33:	// Datenpunkt MotorNumber
		CAN_Index:=16#26C9;
		CAN_Subindex:=16#0;
		CAN_Length:=16#1;
		CAN_RW_Mode:=1;
		CAN_ScaleNum:=1;
		CAN_ScaleDenum:=1;
		CAN_ScaleOffset:=0;
		CAN_Description:='MotorNumber';
		CAN_Unit:='-';
		CAN_Datatype:=8;
		iDpAddres:=ADR(iMotorNumber);
		
		IF bReadSuccesfull THEN
			stPumpInformation.iMotorNumber:=iMotorNumber;
			stPumpinformation.arrPumpInformation[State_CAN].sValue:=USINT_TO_STRING(iMotorNumber);
			bReadSuccesfull:=FALSE;	
			State_CAN := State_CAN+1;
		END_IF	
		
	34:	// Datenpunkt CalculatedPressureCorrected
		CAN_Index:=16#26CA;
		CAN_Subindex:=16#0;
		CAN_Length:=16#2;
		CAN_RW_Mode:=1;
		CAN_ScaleNum:=1;
		CAN_ScaleDenum:=10;
		CAN_ScaleOffset:=0;
		CAN_Description:='CalculatedPressureCorrected';
		CAN_Unit:='mWs';
		CAN_Datatype:=13;
		iDpAddres:=ADR(iCalculatedPressureCorrected);
		
		IF bReadSuccesfull THEN
			stPumpInformation.nCalculatedPressureCorrected:=SCALE(iCalculatedPressureCorrected,CAN_ScaleNum,CAN_ScaleDenum,CAN_ScaleOffset);
			stPumpinformation.arrPumpInformation[State_CAN].sValue:=LREAL_TO_STRING(stPumpInformation.nCalculatedPressureCorrected);
			bReadSuccesfull:=FALSE;	
			State_CAN := State_CAN+1;
		END_IF	
		
	35:	// Datenpunkt SperrzeitDPspitzenlast
		CAN_Index:=16#26CB;
		CAN_Subindex:=16#0;
		CAN_Length:=16#1;
		CAN_RW_Mode:=1;
		CAN_ScaleNum:=1;
		CAN_ScaleDenum:=1;
		CAN_ScaleOffset:=0;
		CAN_Description:='SperrzeitDPspitzenlast';
		CAN_Unit:='s';
		CAN_Datatype:=8;
		iDpAddres:=ADR(iSperrzeitDPspitzenlast);
		
		IF bReadSuccesfull THEN
			stPumpInformation.iSperrzeitDPspitzenlast:=iSperrzeitDPspitzenlast;
			stPumpinformation.arrPumpInformation[State_CAN].sValue:=USINT_TO_STRING(iSperrzeitDPspitzenlast);
			bReadSuccesfull:=FALSE;	
			State_CAN := State_CAN+1;
		END_IF		

	36:	// Datenpunkt E255Index
		CAN_Index:=16#26CC;
		CAN_Subindex:=16#1;
		CAN_Length:=16#2;
		CAN_RW_Mode:=1;
		CAN_ScaleNum:=1;
		CAN_ScaleDenum:=1;
		CAN_ScaleOffset:=0;
		CAN_Description:='E255Index';
		CAN_Unit:='-';
		CAN_Datatype:=9;
		iDpAddres:=ADR(iE255Index);
		
		IF bReadSuccesfull THEN
			stPumpInformation.iE255Index:=iE255Index;
			stPumpinformation.arrPumpInformation[State_CAN].sValue:=UINT_TO_STRING(iE255Index);
			bReadSuccesfull:=FALSE;	
			State_CAN := State_CAN+1;
		END_IF	
		
	37:	// Datenpunkt E255Value
		CAN_Index:=16#26CD;
		CAN_Subindex:=16#1;
		CAN_Length:=16#1;
		CAN_RW_Mode:=1;
		CAN_ScaleNum:=1;
		CAN_ScaleDenum:=1;
		CAN_ScaleOffset:=0;
		CAN_Description:='E255Value';
		CAN_Unit:='-';
		CAN_Datatype:=8;
		iDpAddres:=ADR(iE255Value);
		
		IF bReadSuccesfull THEN
			stPumpInformation.iE255Value:=iE255Value;
			stPumpinformation.arrPumpInformation[State_CAN].sValue:=USINT_TO_STRING(iE255Value);
			bReadSuccesfull:=FALSE;	
			State_CAN := State_CAN+1;
		END_IF		
		
	38:	// Datenpunkt FUlimits
		CAN_Index:=16#26CE;
		CAN_Subindex:=16#1;
		CAN_Length:=16#1;
		CAN_RW_Mode:=1;
		CAN_ScaleNum:=1;
		CAN_ScaleDenum:=1;
		CAN_ScaleOffset:=0;
		CAN_Description:='FUlimits';
		CAN_Unit:='-';
		CAN_Datatype:=8;
		iDpAddres:=ADR(iFUlimits);
		
		IF bReadSuccesfull THEN
			stPumpInformation.iFUlimits:=iFUlimits;
			stPumpinformation.arrPumpInformation[State_CAN].sValue:=USINT_TO_STRING(iFUlimits);
			bReadSuccesfull:=FALSE;	
			State_CAN := State_CAN+1;
		END_IF				
*)		
		
	39:	// Datenpunkt BusCommand
		iBusCommand:=INT_TO_USINT(stPumpInformation.eBusCommand);
		
		CAN_Index:=16#200A;
		CAN_Subindex:=16#0;
		CAN_Length:=16#1;
		CAN_RW_Mode:=2;
		
		MEMCPY(ADR(CAN_WriteData),ADR(iBusCommand),CAN_Length);
	
	40: // Datenpunkt BusControlMode
		iBusControlMode:=INT_TO_USINT(stPumpInformation.eBusControlMode);

		CAN_Index:=16#2009;
		CAN_Subindex:=16#0;
		CAN_Length:=16#1;
		CAN_RW_Mode:=2;
		
		MEMCPY(ADR(CAN_WriteData),ADR(iBusControlMode),CAN_Length);	
		
	41: // Datenpunkt BusSetpoint
		CAN_Index:=16#2008;
		CAN_Subindex:=16#0;
		CAN_Length:=16#2;
		CAN_RW_Mode:=2;		

		IF bUseAbsoluteSetpoint AND imaxValue<>0 THEN
			iBusSetpoint:=LREAL_TO_INT (SCALE(stPumpInformation.nBusSetpoint/stPumpInformation.nmaxValue*100,100,1,0));
		ELSE
			iBusSetpoint:=LREAL_TO_INT (SCALE(stPumpInformation.nBusSetpoint,100,1,0));
		END_IF
				
		MEMCPY(ADR(CAN_WriteData),ADR(iBusSetpoint),CAN_Length);
		
	42: // Step to First DP
		CAN_RW_Mode:=0;
		State_CAN := 1;
	END_CASE
	
// SDO_Datenpunkte lesen/schreiben
	CASE CAN_RW_Mode OF
	0:  // Bausteine nicht ausführen		
	1:	// SDO_Read
		CAN_SDO_READ(
			StartReading := CAN_Start,
			CO_Index := 	CAN_Index,
			CO_SubIndex := 	CAN_Subindex,
			DataLength := 	CAN_Length,
			PortNr := 		CAN_NodePort,
			ADSNetID :=		sCAN_NetID,
(*			ScaleNum :=		CAN_ScaleNum,
			ScaleDenum := 	CAN_ScaleDenum,
			ScaleOffset := 	CAN_ScaleOffset*)
			);
			
		IF CAN_Start THEN
			IF CAN_SDO_READ.ReadDataAvailable THEN
				CAN_ReadError := CAN_SDO_READ.Error;
				IF CAN_SDO_READ.Error<>0  THEN
					iReadError:=iReadError+1;
					stPumpinformation.arrPumpInformation[State_CAN].bReadSuccesfull:=FALSE;
					stPumpinformation.arrPumpInformation[State_CAN].sDatapointNo:=CONCAT (DWORD_TO_HEXSTR(CAN_Index,2,FALSE),CONCAT('_',DWORD_TO_HEXSTR(CAN_Subindex,2,FALSE)));
					stPumpinformation.arrPumpInformation[State_CAN].sDescription:=CAN_Description;
					stPumpinformation.arrPumpInformation[State_CAN].sUnit:=CAN_Unit;		
					stPumpinformation.arrPumpInformation[State_CAN].eDatatyp:=CAN_Datatype;	
					State_CAN := State_CAN+1;
				ELSE
					CAN_ReadData := CAN_SDO_READ.ReadData;
					MEMCPY(iDpAddres,ADR(CAN_ReadData),CAN_Length);
					stPumpinformation.arrPumpInformation[State_CAN].bReadSuccesfull:=TRUE;
					stPumpinformation.arrPumpInformation[State_CAN].sDatapointNo:=CONCAT (DWORD_TO_HEXSTR(CAN_Index,2,FALSE),CONCAT('_',DWORD_TO_HEXSTR(CAN_Subindex,2,FALSE)));
					stPumpinformation.arrPumpInformation[State_CAN].sDescription:=CAN_Description;
					stPumpinformation.arrPumpInformation[State_CAN].sUnit:=CAN_Unit;		
					stPumpinformation.arrPumpInformation[State_CAN].eDatatyp:=CAN_Datatype;				
					bReadSuccesfull:=TRUE;	
				END_IF		
				CAN_Start := FALSE;
				CAN_RW_Mode:=0;
			END_IF
		ELSE
			CAN_Start:=TRUE;
		END_IF

			
	2: 	// SDO_Write
		IF bReadOnly THEN
			State_CAN := 1;
			CAN_Start:=FALSE;
		ELSE
			CAN_SDO_WRITE(
				StartWriting := CAN_Start,
				CO_Index := 	CAN_Index,
				CO_SubIndex := 	CAN_Subindex,
				DataLength := 	CAN_Length,
				PortNr := 		CAN_NodePort,
				ADSNetID:=		sCAN_NetID,
				WriteData:= 	CAN_WriteData
				);			
			IF CAN_Start THEN
				IF CAN_SDO_WRITE.WriteDataFinished THEN
					CAN_WriteError := CAN_SDO_WRITE.Error;
					IF CAN_SDO_Write.Error<>0  THEN
						iWriteError:=iWriteError+1;
					END_IF
					CAN_Start := FALSE;
					State_CAN := State_CAN+1;
				END_IF
			ELSE
				CAN_Start:=TRUE;
			END_IF
		END_IF			
	END_CASE

// Structure
	(*stPumpInformation.iSpeed:= iSpeed;
	stPumpInformation.nPressure:= nPressure;
	stPumpInformation.nFlow:= nFlow;
	stPumpInformation.nInputPower:= nInputPower;
	stPumpInformation.nConsumption:= nConsumption;
	stPumpInformation.nMediumTemp:= nMediumTemp;
	stPumpInformation.nOperatingHours:= nOperatingHours;
	stPumpInformation.eEff_Command:= eEff_Command;
	stPumpInformation.eEff_ControlMode:= eEff_ControlMode;
	stPumpInformation.nEff_Setpoint:= nEff_Setpoint;
	stPumpInformation.nEff_Setpoint_abs:= nEff_Setpoint_abs;
	stPumpInformation.eSel_Command:=eSel_Command;							
	stPumpInformation.eSel_ControlMode:=eSel_ControlMode;							
	stPumpInformation.nSel_Setpoint:=nSel_Setpoint;
	stPumpInformation.nSel_Setpoint_abs:=nSel_Setpoint_abs;					
	stPumpInformation.iPumpType:= iPumpType;
	stPumpInformation.nMaxValue:= nMaxValue;
	stPumpInformation.iCurrentWarning:= iCurrentWarning;*)


// Write Datapoints to LogArray
	iDatapoints_Pump:=0;
	arrDatenpunkt_IDs_Pump[iDatapoints_Pump]:='iSpeed	[rpm]';
	arrDatenpunkt_Values_Pump[iDatapoints_Pump]:=UINT_TO_STRING(stPumpInformation.iSpeed);
	iDatapoints_Pump:=iDatapoints_Pump+1;
		
	arrDatenpunkt_IDs_Pump[iDatapoints_Pump]:='nPressure	[mWs]';
	arrDatenpunkt_Values_Pump[iDatapoints_Pump]:=LREAL_TO_FMTSTR(stPumpInformation.nPressure,2,TRUE);
	iDatapoints_Pump:=iDatapoints_Pump+1;

	arrDatenpunkt_IDs_Pump[iDatapoints_Pump]:='nFlow	[m³/h]';
	arrDatenpunkt_Values_Pump[iDatapoints_Pump]:=LREAL_TO_FMTSTR(stPumpInformation.nFlow,1,TRUE);
	iDatapoints_Pump:=iDatapoints_Pump+1;		
	
	arrDatenpunkt_IDs_Pump[iDatapoints_Pump]:='nInputPower	[W]';
	arrDatenpunkt_Values_Pump[iDatapoints_Pump]:=LREAL_TO_FMTSTR(stPumpInformation.nInputPower,1,TRUE);
	iDatapoints_Pump:=iDatapoints_Pump+1;
	
	arrDatenpunkt_IDs_Pump[iDatapoints_Pump]:='nConsumption	[kWh]';
	arrDatenpunkt_Values_Pump[iDatapoints_Pump]:=LREAL_TO_FMTSTR(stPumpInformation.nConsumption,0,TRUE);
	iDatapoints_Pump:=iDatapoints_Pump+1;
	
	arrDatenpunkt_IDs_Pump[iDatapoints_Pump]:='iPressureSensorSource	[°-]';
	arrDatenpunkt_Values_Pump[iDatapoints_Pump]:=USINT_TO_STRING(stPumpInformation.iPressureSensorSource);
	iDatapoints_Pump:=iDatapoints_Pump+1;
	
	arrDatenpunkt_IDs_Pump[iDatapoints_Pump]:='nOperatingHours	[h]';
	arrDatenpunkt_Values_Pump[iDatapoints_Pump]:=LREAL_TO_FMTSTR(stPumpInformation.nOperatingHours,0,TRUE);
	iDatapoints_Pump:=iDatapoints_Pump+1;
	
	arrDatenpunkt_IDs_Pump[iDatapoints_Pump]:='eEff_Command	[]';
	arrDatenpunkt_Values_Pump[iDatapoints_Pump]:=INT_TO_STRING(stPumpInformation.eEff_Command);
	iDatapoints_Pump:=iDatapoints_Pump+1;
	
	arrDatenpunkt_IDs_Pump[iDatapoints_Pump]:='eEff_ControlMode	[]';
	arrDatenpunkt_Values_Pump[iDatapoints_Pump]:=INT_TO_STRING(stPumpInformation.eEff_ControlMode);
	iDatapoints_Pump:=iDatapoints_Pump+1;
	
	arrDatenpunkt_IDs_Pump[iDatapoints_Pump]:='nEff_Setpoint	[%]';
	arrDatenpunkt_Values_Pump[iDatapoints_Pump]:=LREAL_TO_FMTSTR(stPumpInformation.nEff_Setpoint,2,TRUE);
	iDatapoints_Pump:=iDatapoints_Pump+1;
	
	arrDatenpunkt_IDs_Pump[iDatapoints_Pump]:='nEff_Setpoint_abs	[rpm, mWs]';
	arrDatenpunkt_Values_Pump[iDatapoints_Pump]:=LREAL_TO_FMTSTR(stPumpInformation.nEff_Setpoint_abs,2,TRUE);
	iDatapoints_Pump:=iDatapoints_Pump+1;

	arrDatenpunkt_IDs_Pump[iDatapoints_Pump]:='eSel_Command	[]';
	arrDatenpunkt_Values_Pump[iDatapoints_Pump]:=INT_TO_STRING(stPumpInformation.eSel_Command);
	iDatapoints_Pump:=iDatapoints_Pump+1;
	
	arrDatenpunkt_IDs_Pump[iDatapoints_Pump]:='eSel_ControlMode	[]';
	arrDatenpunkt_Values_Pump[iDatapoints_Pump]:=INT_TO_STRING(stPumpInformation.eSel_ControlMode);
	iDatapoints_Pump:=iDatapoints_Pump+1;
	
	arrDatenpunkt_IDs_Pump[iDatapoints_Pump]:='nSel_Setpoint	[%]';
	arrDatenpunkt_Values_Pump[iDatapoints_Pump]:=LREAL_TO_FMTSTR(stPumpInformation.nSel_Setpoint,2,TRUE);
	iDatapoints_Pump:=iDatapoints_Pump+1;
	
	arrDatenpunkt_IDs_Pump[iDatapoints_Pump]:='nSel_Setpoint_abs	[rpm, mWs]';
	arrDatenpunkt_Values_Pump[iDatapoints_Pump]:=LREAL_TO_FMTSTR(stPumpInformation.nSel_Setpoint_abs,2,TRUE);
	iDatapoints_Pump:=iDatapoints_Pump+1;
	
	arrDatenpunkt_IDs_Pump[iDatapoints_Pump]:='iPumpType	[]';
	arrDatenpunkt_Values_Pump[iDatapoints_Pump]:=UINT_TO_STRING(stPumpInformation.iPumpType);
	iDatapoints_Pump:=iDatapoints_Pump+1;
	
	arrDatenpunkt_IDs_Pump[iDatapoints_Pump]:='nMaxValue	[rpm, mWs]';
	arrDatenpunkt_Values_Pump[iDatapoints_Pump]:=LREAL_TO_FMTSTR(stPumpInformation.nMaxValue,0,TRUE);
	iDatapoints_Pump:=iDatapoints_Pump+1;

	arrDatenpunkt_IDs_Pump[iDatapoints_Pump]:='iCurrentWarning	[]';
	arrDatenpunkt_Values_Pump[iDatapoints_Pump]:=USINT_TO_STRING(stPumpInformation.iCurrentWarning);
	iDatapoints_Pump:=iDatapoints_Pump+1;
	
	arrDatenpunkt_IDs_Pump[iDatapoints_Pump]:='iBusStatus	[]';
	arrDatenpunkt_Values_Pump[iDatapoints_Pump]:=USINT_TO_STRING(stPumpInformation.iBusStatus);
	iDatapoints_Pump:=iDatapoints_Pump+1;
	
	arrDatenpunkt_IDs_Pump[iDatapoints_Pump]:='iControlStatus	[]';
	arrDatenpunkt_Values_Pump[iDatapoints_Pump]:=USINT_TO_STRING(stPumpInformation.iControlStatus);
	iDatapoints_Pump:=iDatapoints_Pump+1;
	
	arrDatenpunkt_IDs_Pump[iDatapoints_Pump]:='iReadyForOperation	[]';
	arrDatenpunkt_Values_Pump[iDatapoints_Pump]:=USINT_TO_STRING(stPumpInformation.iReadyForOperation);
	iDatapoints_Pump:=iDatapoints_Pump+1;
	
	arrDatenpunkt_IDs_Pump[iDatapoints_Pump]:='iPumpIsOperating	[]';
	arrDatenpunkt_Values_Pump[iDatapoints_Pump]:=USINT_TO_STRING(stPumpInformation.iPumpIsOperating);
	iDatapoints_Pump:=iDatapoints_Pump+1;
	
	arrDatenpunkt_IDs_Pump[iDatapoints_Pump]:='iServiceRequired	[]';
	arrDatenpunkt_Values_Pump[iDatapoints_Pump]:=USINT_TO_STRING(stPumpInformation.iServiceRequired);
	iDatapoints_Pump:=iDatapoints_Pump+1;
	
	arrDatenpunkt_IDs_Pump[iDatapoints_Pump]:='nElectricalCurrent	[A]';
	arrDatenpunkt_Values_Pump[iDatapoints_Pump]:=LREAL_TO_FMTSTR(stPumpInformation.nElectricalCurrent,2,TRUE);
	iDatapoints_Pump:=iDatapoints_Pump+1;
	
	arrDatenpunkt_IDs_Pump[iDatapoints_Pump]:='nVoltageLevel	[V]';
	arrDatenpunkt_Values_Pump[iDatapoints_Pump]:=LREAL_TO_FMTSTR(stPumpInformation.nVoltageLevel,2,TRUE);
	iDatapoints_Pump:=iDatapoints_Pump+1;

IF bReadOnly THEN	
	arrDatenpunkt_IDs_Pump[iDatapoints_Pump]:='';
	arrDatenpunkt_Values_Pump[iDatapoints_Pump]:='';
	iDatapoints_Pump:=iDatapoints_Pump+1;

	arrDatenpunkt_IDs_Pump[iDatapoints_Pump]:='';
	arrDatenpunkt_Values_Pump[iDatapoints_Pump]:='';
	iDatapoints_Pump:=iDatapoints_Pump+1;
	
	arrDatenpunkt_IDs_Pump[iDatapoints_Pump]:='';
	arrDatenpunkt_Values_Pump[iDatapoints_Pump]:='';
	iDatapoints_Pump:=iDatapoints_Pump-2;
	
ELSE
	arrDatenpunkt_IDs_Pump[iDatapoints_Pump]:='eBusCommand	[]';
	arrDatenpunkt_Values_Pump[iDatapoints_Pump]:=INT_TO_STRING(stPumpInformation.eBusCommand);
	iDatapoints_Pump:=iDatapoints_Pump+1;

	arrDatenpunkt_IDs_Pump[iDatapoints_Pump]:='eBusControlMode	[]';
	arrDatenpunkt_Values_Pump[iDatapoints_Pump]:=INT_TO_STRING(stPumpInformation.eBusControlMode);
	iDatapoints_Pump:=iDatapoints_Pump+1;
	
	arrDatenpunkt_IDs_Pump[iDatapoints_Pump]:='nBusSetpoint	[%, rpm, mWs]';
	arrDatenpunkt_Values_Pump[iDatapoints_Pump]:=LREAL_TO_FMTSTR(stPumpInformation.nBusSetpoint,2,TRUE);
	iDatapoints_Pump:=iDatapoints_Pump+1;
END_IF

END_FUNCTION_BLOCK

// CAN/FB_SDO_READ_v0
FUNCTION_BLOCK FB_SDO_READ_v0
VAR_INPUT
	/// The AMSNetID addres of EL6751
	ADSNetID: STRING(23);
	/// This Port No. addresses the CANopen Node (see System Manager) 
	PortNr: WORD;
	/// This is the Index of the CANopen Object Dictionary Entry
	CO_Index: DWORD;
	/// This is the Sub-Index of the CANopen Object Dictionary Entry
	CO_SubIndex: DWORD;
	/// This is the Length of the CANopen Object Dictionary Entry
	DataLength: DWORD;
	/// only reset to FALSE after ReadDataAvailable=TRUE
	StartReading: BOOL;
	ScaleOffset: LREAL := 0;
	ScaleNum: LREAL := 1;
	ScaleDenum: LREAL := 1;
END_VAR
VAR_OUTPUT
	ReadData: ARRAY[0..255] OF BYTE;
	ReadDataAvailable: BOOL;
	Error: DWORD;
	Read_Value: LREAL; // Achtung: Interpretaion für unsigned Integer Werte
END_VAR
VAR
	state: BYTE := 0;
	ADSREAD: ADSREAD;
	Multiplikator: DWORD;
	Counter: INT;
	temp_Value: LREAL;
END_VAR

CASE state OF
0:
	IF StartReading THEN
		ReadDataAvailable := FALSE;
		Error := 0;
		ADSRead(
			NETID:= ADSNetID,
			PORT:= PortNr,
			IDXGRP:= CO_Index,
			IDXOFFS:= CO_SubIndex,
			LEN:= DataLength,
			DESTADDR:= ADR(ReadData),
			READ:= TRUE,
			TMOUT := T#1s
		);
		IF ADSRead.err THEN
			state := 2;
			(*ReadDataAvailable := TRUE;*)
			Error := ADSRead.ErrId;
		ELSE
			state := 1;
		END_IF
	ELSE
		ADSRead(
			NETID:= ADSNetID,
			PORT:= PortNr,
			IDXGRP:= CO_Index,
			IDXOFFS:= CO_SubIndex,
			LEN:= DataLength,
			DESTADDR:= ADR(ReadData),
			READ:= FALSE,
			TMOUT := T#1s
		);
	END_IF

1:
	ADSRead(READ:= FALSE);
	IF ADSRead.err THEN
		state := 2;
		(*ReadDataAvailable := TRUE;*)
		Error := ADSRead.ErrId;
	ELSE
		IF NOT ADSRead.busy THEN
			state := 2;
			(*ReadDataAvailable := TRUE;*)
		END_IF
	END_IF

2: 
	ADSRead(READ:= FALSE);
	ReadDataAvailable := TRUE;
	state := 0;

	(*Daten wieder zusammenfügen_Start*)
	temp_VALUE:=0;
	Multiplikator:=1;
	FOR Counter:=1 TO DWORD_TO_INT(DataLength) BY 1
	DO
		temp_VALUE:=temp_VALUE + ReadData[Counter-1]*Multiplikator;
		Multiplikator:=Multiplikator*16#100;
	END_FOR;
	(*Daten wieder zusammenfügen_Ende*)
	
	Read_Value:=temp_VALUE*ScaleNum/ScaleDenum+ScaleOffset;
END_CASE

END_FUNCTION_BLOCK

// Datenlogger/FB/FB_FILE
FUNCTION_BLOCK FB_FILE
VAR
	// allgemein
	iStateFile_close			:INT;	
	iStateFile_open				:INT;
	
	// Datum der nächsten Minute
	tNextDate					:TIMESTRUCT;
	sNextYear					:T_MaxString;
	sNextMonth					:T_MaxString;
	sNextDay					:T_MaxString;
	sNextHour					:T_MaxString;
	sNextMinute					:T_MaxString;
	sNextSecond					:T_MaxString;
	sNextMillisecond			:T_MaxString;
	sNextSecond_Null			:T_MaxString:='00';
	
	// Zeitstring für Messdatendatei
	fbFormatTimestring			:FB_FormatString;
	bFormatTimestring_error		:BOOL;
	nFormatTimestring_errID		:UDINT;
	
	// Messdatendateiname	
	sFileName					:STRING (19);
	ePath						:E_OpenPath;
	
	// Datei öffnen
	bOpenFile					:BOOL;
	fbFileOpen					:FB_FileOpen;
	iFileOpen_errID				:UDINT;
	nhFileOpen					:UINT;			// Anzahl geöffneter Dateien
	
	// Datei schließen
	bCloseFile					:BOOL;
	fbFileClose					:FB_FileClose;
	iFileClose_errID			:UDINT;
	
	// Referenz tauschen
	bChangeFile					:BOOL;	
END_VAR

VAR_IN_OUT
// ehemals Globale Variablen	
// Time	
	// Time UTC
	tfDate						:T_Filetime;							(*aktuelles Datum UTC*)
	sYear						:T_MaxString;							(*aktuelles Jahr UTC als String*)
	sMonth						:T_MaxString;							(*aktueller Monat UTC als String*)
	sDay						:T_MaxString;							(*aktueller Tag UTC als String*)
	sHour						:T_MaxString;							(*aktuelle Stunde UTC als String*)
	sMinute						:T_MaxString;							(*aktuelle Minute UTC als String*)
	sSecond						:T_MaxString;							(*aktuelle Sekunde UTC als String*)
	sMilliSecond				:T_MaxString;							(*aktulle Millisekunde UTC als String*)

// File and Folder
	// allgemein
	sFolderPath					:T_MaxString;							(*Pfad, zum Messdatenordner*)
	sFilePath					:T_MaxString;							(*Pfad zur Messdatendatei*)
	
	// Statusvariablen der Dateierstellung
	sLastFile_Changed			:T_MaxString;						(*Minute der letzten Änderung des verwedndeten Datenfiles*)
	sLastFile_Opened			:T_MaxString;						(*Minute des letzten geöffneten Datenfiles*)

	// Dateireferenzen	
	hFile						:UINT;									(*Referenz der aktuellen Messdatendatei*)
	hFile_Close					:UINT;									(*Referenz der zu schließenden Messdatendatei*)
	arrhFile_Open				:ARRAY [0..10] OF UINT;					(*Referenz-Array der geöffneten Messdatendatein*)	

// Logging
	//wNextMeasurement			:LWORD;									(*Zeit des nächsten vorgesehenen Loggings*)
	bLogging_activ				:BOOL;									(*Flag; zeigt an, ob gerade Werte geschrieben werden*)	
	
// Errohandling	
	nError_File_Open			:UINT;
	nError_File_Close			:UINT;	
	nError_File_Change			:UINT;	
END_VAR

// Initialisierung --> Öffen einer Datei
IF sLastFile_Opened = '99' AND sFolderPath <> '' THEN
	bOpenFile:=TRUE;
END_IF

// Zeit in einer Minute
	tNextDate:=FILETIME_TO_SYSTEMTIME(F_TranslateFileTimeBias(tfDate,1,TRUE));
	sNextYear	:= DWORD_TO_DECSTR(tNextDate.wYear, 4);
	sNextMonth	:= DWORD_TO_DECSTR(tNextDate.wMonth, 2);
	sNextDay	:= DWORD_TO_DECSTR(tNextDate.wDay, 2);
	sNextHour	:= DWORD_TO_DECSTR(tNextDate.wHour, 2);
	sNextMinute	:= DWORD_TO_DECSTR(tNextDate.wMinute, 2);
	sNextSecond	:= DWORD_TO_DECSTR(tNextDate.wSecond, 2);
	sNextMillisecond := DWORD_TO_DECSTR(tNextDate.wMilliseconds, 3);
	

// neue Datei alle Viertelstunde
IF (sNextMinute = '00'	OR	sNextMinute = '15'	OR	sNextMinute = '30' OR	sNextMinute = '45')
	AND	(((STRING_TO_INT(sLastFile_Opened)<>STRING_TO_INT(sNextMinute))	AND	(STRING_TO_INT(sLastFile_Opened)<60)) OR	(sLastFile_Opened = '98'))	THEN
		bOpenFile:=TRUE;
		sLastFile_Opened:=sNextMinute;
END_IF	

// Referenz des Logfiles jede Viertelstunde tauschen
IF (sMinute = '00'	OR	sMinute = '15'	OR sMinute = '30'	OR	sMinute = '45')
	AND (((STRING_TO_INT (sLastFile_Changed)<>STRING_TO_INT(sMinute))	AND	(STRING_TO_INT (sLastFile_Changed)<60))	OR	sLastFile_Changed = '98')	THEN
		bChangeFile:=TRUE;
		sLastFile_Changed:=sMinute;
END_IF
(*
// neue Datei alle Viertelstunde
IF (sNextMinute = '00' AND (sLastFile_Opened = '45' OR sLastFile_Opened = '98'))
	OR (sNextMinute = '45' AND (sLastFile_Opened = '30' OR sLastFile_Opened = '98'))
	OR (sNextMinute = '30' AND (sLastFile_Opened = '15' OR sLastFile_Opened = '98'))
	OR (sNextMinute = '15' AND (sLastFile_Opened = '00' OR sLastFile_Opened = '98')) THEN
		bOpenFile:=TRUE;
		sLastFile_Opened:=sNextMinute;
END_IF	

// Referenz des Logfiles jede Viertelstunde tauschen
IF (sMinute = '00' AND (sLastFile_Changed = '45' OR sLastFile_Changed = '98'))
	OR (sMinute = '45' AND (sLastFile_Changed = '30' OR sLastFile_Changed = '98'))
	OR (sMinute = '30' AND (sLastFile_Changed = '15' OR sLastFile_Changed = '98'))
	OR (sMinute = '15' AND (sLastFile_Changed = '00' OR sLastFile_Changed = '98')) THEN
		bChangeFile:=TRUE;
		sLastFile_Changed:=sMinute;
END_IF

// manueller Trigger schließen und öffnen einer neuen Datei
IF	bNewFile_manually THEN
	bNewFile_manually:=FALSE;
	bOpenFile:=TRUE;
	sLastFile_Opened:='99';
	sLastFile_Changed:='99';
END_IF
*)	

// Datei öffnen sobald Signal dafür gesetzt wird	
IF bOpenFile THEN
	CASE iStateFile_open OF
	0: // Datei öffnen
		// Zeitstring für neue Datei
		IF sLastFile_Opened='99' THEN
			fbFormatTimestring(
				sFormat	:='%S-%S-%S_%S-%S-%S',
				arg1	:= F_STRING(sYear),
				arg2	:= F_STRING(sMonth),
				arg3	:= F_STRING(sDay),
				arg4	:= F_STRING(sHour),
				arg5	:= F_STRING(sMinute),
				arg6	:= F_STRING(sSecond),
				sOut	=> sFileName,
				bError	=> bFormatTimestring_error,
				nErrId	=> nFormatTimestring_errID
				);
		ELSE
			fbFormatTimestring(
				sFormat	:='%S-%S-%S_%S-%S-%S',
				arg1	:= F_STRING(sNextYear),
				arg2	:= F_STRING(sNextMonth),
				arg3	:= F_STRING(sNextDay),
				arg4	:= F_STRING(sNextHour),
				arg5	:= F_STRING(sNextMinute),
				arg6	:= F_STRING(sNextSecond_Null),
				sOut	=> sFileName,
				bError	=> bFormatTimestring_error,
				nErrId	=> nFormatTimestring_errID
				);
		END_IF
		
		// kompletter Pfad der Messdatendatei erzeugen		
		sFilePath:=CONCAT(sFolderPath,'\');
		sFilePath:=CONCAT(sFilePath,sFileName);
		sFilePath:=CONCAT(sFilePath,'_Messdaten.csv');
		
		// Datei anlegen
		fbFileOpen(
			bExecute:=FALSE,
			);
		
		fbFileOpen(
			sNetID:='',
			sPathName:=sFilePath,
			nMode:=FOPEN_MODEAPPEND,
			ePath:=ePath,
			bExecute:=TRUE,
			tTimeout:=T#5S,
			);
		
		iStateFile_open:=iStateFile_open+1;
	
	1:	// warten bis Funktionsbaustein fertig
		fbFileOpen(
			bExecute:=FALSE,
			);
		IF NOT fbFileOpen.bBusy THEN
			IF fbFileOpen.bError THEN
				nError_File_Open:=nError_File_Open+1;
				iFileOpen_errID:=fbFileOpen.nErrId;
			ELSE
				arrhFile_open[nhFileOpen]:=fbFileOpen.hFile;
				nhFileOpen:=nhFileOpen+1;
					IF sLastFile_Opened='99' THEN
						sLastFile_Opened:='98';
					END_IF
					IF sLastFile_changed='99' THEN // hier muss ich was tun
						bChangeFile:=TRUE;
						sLAstFile_changed:='98';			
					END_IF
				iFileOpen_errID:=fbFileOpen.nErrId;
			END_IF	
			bOpenFile:=FALSE;
			iStateFile_open:=0;
		END_IF
	END_CASE
END_IF

// Datei austauschen
IF bChangeFile AND NOT bLogging_activ THEN
	IF arrhFile_open[nhFileOpen-1] <> hFile   THEN
		IF NOT(arrhFile_open[nhFileOpen-1]=0 OR nhFileOpen=0) THEN
			IF hFile<>0 THEN
				hFile_close:=hFile;
				bCloseFile:=TRUE;
			END_IF
			nhFileOpen:=nhFileOpen-1;	
			hFile:=arrhFile_open[nhFileOpen];
			arrhFile_open[nhFileOpen]:=0;
		ELSE
			nError_File_Change:=nError_File_Change+1;
		END_IF
	END_IF
	bChangeFile:=FALSE;	
END_IF

	
// Datei schließen, wenn eine neue Datei geöffnet wurde, und Referenz ausgetauscht wurde
IF bCloseFile OR (sLastFile_Changed = '97' AND NOT bLogging_activ) THEN
	CASE iStateFile_close OF	
	0:	//Datei schließen
		fbFileClose(
			bExecute:=FALSE,
			);
		fbFileClose(
			sNetId:='',
			hFile:=hFile_Close,
			bExecute:=TRUE,
			tTimeout:=,
			);
		iStateFile_close:=iStateFile_close+1;
	
	1:	// warten bis Funktionsbaustein fertig	
		fbFileClose(
			bExecute:=FALSE,
			);
		IF NOT fbFileClose.bBusy THEN		
			IF fbFileClose.bError THEN
				nError_File_Close:=nError_File_Close+1;
				iFileClose_errID:=fbFileClose.nErrId;
			END_IF
				iFileClose_errID:=fbFileClose.nErrId;
				iStateFile_close:=0;
			IF nhFileOpen=0 THEN	
				bCloseFile:=FALSE;	
				IF sLastFile_Changed='97'  THEN
					sLastFile_Changed:='99';
					sLastFile_Opened:='99';
					hFile:=0;
				END_IF	
			ELSE
				nhFileOpen:=nhFileOpen-1;
				hFile_Close:=arrhFile_Open[nhFileOpen];
				arrhFile_Open[nhFileOpen]:=0;
			END_IF
		END_IF
	END_CASE
END_IF

END_FUNCTION_BLOCK

// Datenlogger/FB/FB_FOLDER
FUNCTION_BLOCK FB_FOLDER
VAR
	// Hauptverzeichnis erzeugen
	ePath						:E_OpenPath;
	bDirectory_created 			:BOOL;	
	fbCreateDirectoty			:FB_CreateDir;
	iDirectory_errID			:UDINT;
	
	// Zeitstring für Unterverzeichnis
	fbFormatTimestring			:FB_FormatString;
	bFormatTimestring_Error		:BOOL;
	nFormatTimestring_errID		:UDINT;
	sFolderName					:STRING(10);	
	
	// Unterverzeichnis erzeugen
	fbCreateFolder				:FB_CreateDir;
	iFolder_errorID				:UDINT;
	iFolderCounter				:UINT;
	bFolder_error				:BOOL;
	sFolderPath_temp			:T_MaxString;
	
	// Datumsvorausschau in  nPrevNextDate Minuten
	nPrevNextDate				:INT:=0;
	tNextDate					:TIMESTRUCT;
	sNextYear					:T_MaxString;
	sNextMonth					:T_MaxString;
	sNextDay					:T_MaxString;
END_VAR

VAR_IN_OUT
// ehemals Globale Variablen
	// General
	sDataPath					:T_MaxString; 							(*Pfad der Messdaten*)
	
	// Time
	tfDate						:T_Filetime;							(*aktuelles Datum UTC*)
	wDate						:LWORD;									(*aktuelles Datum UTC*)
	sYear						:T_MaxString;							(*aktuelles Jahr UTC als String*)	

// File and Folder
	// allgemein
	iStateFolder				:INT;									(*Case Auswahl der Ordnererzeugung*)
	arrLastFolder				:ARRAY [0..2] OF STRING;				(*letzter erzeugter Datumsordner*)
	sFolderPath					:T_MaxString;							(*Pfad, zum Messdatenordner*)

// Errohandling	
	nError_Folder				:UINT;
END_VAR

IF wDate <>0 THEN
	CASE iStateFolder OF
	0:	// Hauptverzeichnis "Messdaten" anlegen
		fbCreateDirectoty(
			bExecute:=FALSE,
			);
			
		// Ordner erzeugen
		fbCreateDirectoty(
			sNetId:='',
			sPathName:=sDataPath,
			ePath:=ePath,
			bExecute:=TRUE,
			tTimeout:=T#5S,
			);		
		iStateFolder:=1;
		
	1:	// warten bis Funktionsbaustein fertig ist
		fbCreateDirectoty(
			bExecute:=FALSE,
			);
		IF NOT fbCreateDirectoty.bBusy THEN
			IF fbCreateDirectoty.bError THEN
				iDirectory_errID:=fbCreateDirectoty.nErrId;
				nError_Folder:=nError_Folder+1;
			END_IF
			iDirectory_errID:=fbCreateDirectoty.nErrId;
			bDirectory_created:=TRUE;
			iStateFolder:=2;
			nPrevNextDate:=0;		
		END_IF
	
	2: // Unterverzeichnis erzeugen
		// checken ob übernächste Minute zu neuem Tag gehört
		tNextDate:=FILETIME_TO_SYSTEMTIME(F_TranslateFileTimeBias(tfDate,nPrevNextDate,TRUE));
		sNextYear	:= DWORD_TO_DECSTR(tNextDate.wYear, 4);
		sNextMonth	:= DWORD_TO_DECSTR(tNextDate.wMonth, 2);
		sNextDay	:= DWORD_TO_DECSTR(tNextDate.wDay, 2);
		
		// neuen Ordner um 23:58 UHR anlegen
		IF sNextDay <> arrLastFolder[0]
				OR sNextMonth <> arrLastFolder[1]
				OR sNextYear <> arrLastFolder[2] AND sYear<>''  THEN
		
			arrLastFolder[0]:=sNextDay;
			arrLastFolder[1]:=sNextMonth;
			arrLastFolder[2]:=sNextYear;
		
			// Zeitsting für Unterverzeichnis bauen
			fbFormatTimestring(
					sFormat	:= '%S-%S-%S',
					arg1	:= F_STRING(sNextYear),
					arg2	:= F_STRING(sNextMonth),
					arg3	:= F_STRING(sNextDay),
					sOut	=> sFolderName,
					bError	=> bFormatTimestring_error,
					nErrId	=> nFormatTimestring_errID
			);
			
			// Pfad für Messdatendatei speichern		
			sFolderPath_temp:=CONCAT(sDataPath,sFolderName);
			
			fbCreateFolder(
			bExecute:=FALSE,);
			
			// Verzeichnis erzeugen
			fbCreateFolder(
				sNetId:='',
				sPathName:=sFolderPath_temp,
				ePath:=ePath,
				bExecute:=TRUE,
				tTimeout:=T#5S,
			);	
			iStateFolder:=3;
		END_IF
	
	3:	// warten bis FB fertig, Übergabe Ordnerpfad
		fbCreateFolder(
			bExecute:=FALSE,
			);	
		IF NOT fbCreateFolder.bBusy THEN
			bFolder_error:=fbCreateFolder.bError;
			iFolder_errorID:=fbCreateFolder.nErrId;
			IF bFolder_error THEN
				nError_Folder:=nError_Folder+1;
			END_IF
			sFolderPath:=sFolderPath_temp;
			iStateFolder:=2;
			nPrevNextDate:=2;
		END_IF		
	END_CASE
END_IF

END_FUNCTION_BLOCK

// Datenlogger/FB/FB_LOGGING
FUNCTION_BLOCK FB_LOGGING
VAR
	// allgemien
	iStateLogging				:INT;	
	arrTMAXempty				:ARRAY [0..499] OF T_MaxString;			// Empty Array to Reset Array

	// Zeitsteuerung Speicherzyklus
	Timer_Logging				:TON;
	bTimer_trigger				:BOOL:=TRUE;
	bLogging					:BOOL;
	
	// Zeitstempel bauen
	fbFormatTimestamp			:FB_FormatString;
	bFormatTimestamp_error		:BOOL;
	nFormatTimestamp_errID		:UDINT;
	sMeasurement_time			:T_MaxString;
	sMeasurement_date			:T_MaxString;
	sLMeasurement_time			:T_MaxString;
	sLMeasurement_date			:T_MaxString;
	
	// Messstring bauen
	fbFormatMeasString			:FB_FormatString;
	bFormatMeasString_error		:BOOL;
	nFormatMeasString_errID		:UDINT;
	sDelimiter					:T_MaxString:='$09';		(*$09 = Tab stop*)
	sSpaces						:T_MaxString:='$20';		(*$20 = Leerzeichen*)
	iDatapoint_log				:INT:=0;
	
	// Datenpunktstring temporär
	sMeasString_temp			:T_MaxString;

	// Puffer der Messdaten
	arrDP_ID_buffer				:ARRAY [0..499] OF T_MaxString;			(*Puffer der Beschreibung/ID der Datenpunkte*)
	arrDP_Value_buffer			:ARRAY [0..499] OF T_MaxString;			(*Puffer Messwerte der Datenpunkte*)
	iBuffer						:INT;
	
	// Store Meta Information
	bStoreMetaDataInFile		:BOOL:=TRUE;	// Flag to activate MetaLogging
END_VAR
VAR PERSISTENT	
	arrMetaID					:ARRAY [0..499] OF T_MaxString;			// Array of logged MetaIDs
	sLastMetaDay			:T_MaxString;								// Stored Day to Reset MetaIDs
END_VAR
VAR							
//	arrBuffer					:ARRAY [0..99] OF Log_Datapoint;
	iMetaID						:INT;									// StateVariable to Compare MetaIDs
	iMeta						:INT;									// Row of Meta Data To Store
	arrMetaData					:ARRAY [0..499] OF Log_Datapoint;		// MetaDataToStore
//	bStoreMeta					:BOOL;
	iMetaBuffer					:INT;									// stateVariable to write MetaData into Buffer
	arrMetaDataBuffer			:ARRAY [0..499] OF Log_Datapoint;		// MetaData Buffer
	arrMetaDataEmpty			:ARRAY [0..499] OF Log_Datapoint;		// Empty Struct to Reset MetaData Struct
	
	// MetaFileHandling
	iState_StoreMeta		:INT;
	sMetaFileName			:T_MaxString:='_MetaData.txt';	

	sFilePathMeta			:T_MaxString;
	fbFileOpenMeta			:FB_FileOpen;
	iFileOpenMeta_errID		:UDINT;
	hFileMeta				:UINT;
	fbFileCloseMeta			:FB_FileClose;
	iFileCloseMeta_errID	:UDINT;
	
	// Meta WriteToFile
	iMetaInfo				:INT;	
	sStringMeta				:T_MaxString;
	fbFilePutsMeta			:FB_FilePuts;
	iFilePutsMeta_errID		:UDINT;
	bPutsMeta_busy			:BOOL;
	bPutsMeta_error			:BOOL;
	iPutsMeta_errorID		:UDINT;
	nErrorMeta_LogError		:INT;

//	bResetMetaID			:BOOL;
	

//	fbFormatMetaFilepath			:FB_FormatString;
//	bFormatMetaFilepath_error		:BOOL;
//	nFormatMetaFilepath_errID		:UDINT;	
	
		
	// Datenpunktstring für schreiben vorbereiten
	fb_CSVbuffer				:FB_CSVMemBufferWriter;
	eCmd    					:E_EnumCmdType := eEnumCmd_First;
	putValue 					:T_MaxString ;
	pValue  					:POINTER TO BYTE := 0;
	cbValue  					:UDINT := 0;
	bCRLF   					:BOOL :=TRUE;
	pBuffer  					:POINTER TO BYTE;
	cbBuffer 					:UDINT;
	iSize_buffer				:UDINT;

	// Datenpunktstring
	sMeasString					:T_MaxString;

	// Datenpunktstring schreiben
    fbFilePuts       			:FB_FilePuts;
	bPuts_busy					:BOOL;
	bPuts_error					:BOOL;
	iPuts_errorID				:UDINT;

	// Messzyklus
	tfNextMeasurement			:T_Filetime;
	tNextMeasurement			:TIMESTRUCT;
	bStoreData_to_buffer		:BOOL;
	
	// Watchdog Datenpunkte schreiben
	bWatchdogDPwrite			:BOOL;
	fbWatchdogDPwrite			:TON;
	tWatchdogDPwrite_Time		:TIME;
END_VAR
VAR_OUTPUT
	// information of Loged Datapoints
	iNumberOfLoggedDP 			:INT;
	arrLoggedDatapoints			:ARRAY [0..499] OF Log_Datapoint;		(*Array of Logged Datapoints*)
END_VAR
VAR_IN_OUT
// ehemals Globale Variablen
// General	
	arrLogDatapoints			:ARRAY [0..499] OF Log_Datapoint;		(*Logging Input*)
	bArrayStored				:BOOL;
//	arrDatapoint_ID				:ARRAY [0..99] OF T_MaxString;			(*Beschreibung der Datenpunkte*)
//	arrDatapoint_Value			:ARRAY [0..99] OF T_MaxString;			(*Messwerte der Datenpunkte*)
//	sDataPath					:T_MaxString:='C:\Messdaten\'; 			(*Pfad der Messdaten*)
	tLogCycleTime				:TIME;									(*Messzyklusvorgabe*)
	
// Time	
//	bUseTcTime					:BOOL;									(*Zeitbasis: fortlaufende TwinCAT-Uhr initialisiert durch Windows*)
	// Time local
//	tLDate						:TIMESTRUCT;							(*aktuelles Datum lokal*)
//	tfLDate						:T_Filetime;							(*aktuelles Datum lokal*)
	sLYear						:T_MaxString;							(*aktuelles Jahr lokal als String*)
	sLMonth						:T_MaxString;							(*aktueller Monat lokal als String*)
	sLDay						:T_MaxString;							(*aktueller Tag lokal als String*)
	sLHour						:T_MaxString;							(*aktuelle Stunde lokal als String*)
	sLMinute					:T_MaxString;							(*aktuelle Minute lokal als String*)
	sLSecond					:T_MaxString;							(*aktuelle Sekunde lokal als String*)
	sLMilliSecond				:T_MaxString;							(*aktulle Millisekunde lokal als String*)
	// Time UTC
//	tDate						:TIMESTRUCT;							(*aktuelles Datum UTC*)
//	tfDate						:T_Filetime;							(*aktuelles Datum UTC*)
	wDate						:LWORD;									(*aktuelles Datum UTC*)
	sYear						:T_MaxString;							(*aktuelles Jahr UTC als String*)
	sMonth						:T_MaxString;							(*aktueller Monat UTC als String*)
	sDay						:T_MaxString;							(*aktueller Tag UTC als String*)
	sHour						:T_MaxString;							(*aktuelle Stunde UTC als String*)
	sMinute						:T_MaxString;							(*aktuelle Minute UTC als String*)
	sSecond						:T_MaxString;							(*aktuelle Sekunde UTC als String*)
	sMilliSecond				:T_MaxString;							(*aktulle Millisekunde UTC als String*)

// File and Folder
	// allgemein
	sFolderPath					:T_MaxString;							(*Pfad, zum Messdatenordner*)
	// Dateireferenzen	
	hFile						:UINT;									(*Referenz der aktuellen Messdatendatei*)	
	
// Logging
	wNextMeasurement			:LWORD;									(*Zeit des nächsten vorgesehenen Loggings*)
	bLogging_activ				:BOOL;									(*Flag; zeigt an, ob gerade Werte geschrieben werden*)
	bLogUtcTime					:BOOL;									(*UTC Zeit mitloggen*)
	bLogLocalTime				:BOOL;									(*lokale Zeit mitloggen*)
	bOldOutputFile				:BOOL;									(*FALSE(default)OutputFile:"idTABvalue"; TRUE(oldFormat):OutputFile: "DescriptionTAB[unit]TABvalue"*)
	
// Errohandling
	nError_Logging				:UINT;	
	nError_Datalogger			:UINT;
END_VAR

// Initialisierung
IF ((wNextMeasurement=0) OR (wDate>wNextMeasurement+2*10000*TIME_TO_WORD(tLogCycleTime)) OR (wDate<wNextMeasurement-2*10000*TIME_TO_WORD(tLogCycleTime))) AND wDate <> 0 THEN
	wNextMeasurement:=wDate;
END_IF

IF bOldOutputFile THEN
	bStoreMetaDataInFile:=FALSE;
ELSE
	bStoreMetaDataInFile:=TRUE;
END_IF

// Zeitsteuerung
IF wDate >= wNextMeasurement AND NOT bLogging_activ AND wNextMeasurement > 0 THEN
	wNextMeasurement:=wNextMeasurement+10000*TIME_TO_WORD(tLogCycleTime);
	MEMCPY(ADR(tfNextMeasurement.dwHighDateTime),ADR(wNextMeasurement)+4,4);
	MEMCPY(ADR(tfNextMeasurement.dwLowDateTime),ADR(wNextMeasurement),4);
	tNextMeasurement:=FILETIME_TO_SYSTEMTIME(tfNextMeasurement);
	bLogging:=TRUE;
	bStoreData_to_buffer:=TRUE;
END_IF	

IF sDay<>sLastMetaDay THEN
	arrMetaID:=arrTMAXempty;
	sLastMetaDay:=sDay;
END_IF

// Datenpunkte zum Messzeitpunkt im Buffer zwischenspeichern
IF bStoreData_to_buffer THEN
	bArrayStored:=TRUE;
	bStoreData_to_buffer:=FALSE;
	(*String für Messzeit UTC*)
	fbFormatTimestamp(
		sFormat	:= '%S:%S:%S.%S',
		arg1	:= F_STRING(sHour),
		arg2	:= F_STRING(sMinute),
		arg3	:= F_STRING(sSecond),
		arg4:= F_STRING(sMilliSecond),
		sOut	=> sMeasurement_time,
		bError	=> bFormatTimestamp_error,
		nErrId	=> nFormatTimestamp_errID
	);

	(*String für Messdatum UTC*)
	fbFormatTimestamp(
		sFormat	:= '%S-%S-%S',
		arg1	:= F_STRING(sYear),
		arg2	:= F_STRING(sMonth),
		arg3	:= F_STRING(sDay),
		sOut	=> sMeasurement_date,
		bError	=> bFormatTimestamp_error,
		nErrId	=> nFormatTimestamp_errID
	);
	
	IF bFormatTimestamp_error THEN
		nError_Logging:=nError_Logging+1;
	END_IF
	
	(*String für Messzeit lokal*)
	fbFormatTimestamp(
		sFormat	:= '%S:%S:%S.%S',
		arg1	:= F_STRING(sLHour),
		arg2	:= F_STRING(sLMinute),
		arg3	:= F_STRING(sLSecond),
		arg4:= F_STRING(sLMilliSecond),
		sOut	=> sLMeasurement_time,
		bError	=> bFormatTimestamp_error,
		nErrId	=> nFormatTimestamp_errID
	);

	IF bFormatTimestamp_error THEN
		nError_Logging:=nError_Logging+1;
	END_IF
	
	(*String für Messdatum loakl*)
	fbFormatTimestamp(
		sFormat	:= '%S-%S-%S',
		arg1	:= F_STRING(sLYear),
		arg2	:= F_STRING(sLMonth),
		arg3	:= F_STRING(sLDay),
		sOut	=> sLMeasurement_date,
		bError	=> bFormatTimestamp_error,
		nErrId	=> nFormatTimestamp_errID
	);
	
	IF bFormatTimestamp_error THEN
		nError_Logging:=nError_Logging+1;
	END_IF
	
	eCmd:= eEnumCmd_First;
	
	(*alle Messwete zum akutellen Zeitpunkt im Puffer speichern*)
(*	(*Puffer alt, zwei Arrays*)
	arrDP_ID_buffer:=arrDatapoint_ID;
	arrDP_Value_buffer:=arrDatapoint_Value;
*)
	(* Puffer neu --> eine Struct *)
	// bei zeitlichen Problemen auf mehrere Zykeln aufteilen
	arrLoggedDatapoints:=arrLogDatapoints;
	FOR iBuffer:=0 TO 499 BY 1 DO
		IF arrLogDatapoints[iBuffer].sDescription<>'' OR arrLogDatapoints[iBuffer].sID <>'' THEN
			arrDP_Value_buffer[iBuffer]:=arrLogDatapoints[iBuffer].sValue;
			IF arrLogDatapoints[iBuffer].sDescription = '' THEN
				arrLogDatapoints[iBuffer].sDescription:=arrLogDatapoints[iBuffer].sID;
			END_IF		
	
			IF NOT bOldOutputFile THEN (*Puffer füllen*)
				IF arrLogDatapoints[iBuffer].sID<>'' THEN
					arrDP_ID_buffer[iBuffer]:=arrLogDatapoints[iBuffer].sID;
				ELSE
					arrDP_ID_buffer[iBuffer]:=arrLogDatapoints[iBuffer].sDescription;
				END_IF
			ELSE (* Puffer füllen für altes Ausgabeformat füllen*)
				arrDP_ID_buffer[iBuffer]:=CONCAT(arrLogDatapoints[iBuffer].sDescription,'$09[');
				IF arrLogDatapoints[iBuffer].sUnit<>'' THEN
					arrDP_ID_buffer[iBuffer]:=CONCAT(arrDP_ID_buffer[iBuffer],arrLogDatapoints[iBuffer].sUnit);
				ELSE
					arrDP_ID_buffer[iBuffer]:=CONCAT(arrDP_ID_buffer[iBuffer],'-');
				END_IF
				arrDP_ID_buffer[iBuffer]:=CONCAT(arrDP_ID_buffer[iBuffer],']');
			END_IF
					
